# B&R Automation Studio project Kesim (part 2)

#### FbFileCreate.st - File oluşturur.
```iecst
(********************************************************************
 * COPYRIGHT --  B&R Industrial Automation GmbH
 ********************************************************************
 * Library: aLibFile
 * Function Block: FbFileCreate
 * Author: kay3a
 * Created: August 27, 2024/4:58 PM
 ********************************************************************
 * Description: Bu FB secili DeviceName altinda bulunan foler içerisine file olusturur.
 ********************************************************************)
FUNCTION_BLOCK FbFileCreate

	//|ŻŻŻŻŻŻŻŻŻŻŻŻŻŻŻŻŻŻŻŻŻŻŻŻŻŻŻŻŻŻŻŻŻŻŻŻŻŻŻŻŻŻŻŻŻŻŻŻŻŻŻŻŻŻŻŻŻŻŻŻŻŻŻŻŻŻŻŻŻŻŻŻŻ
	//|               FB ENABLE KONTROLU
	//|_________________________________________________________________________

	(* Enable gelirse FB aktiftir. Gelmiyorsa aktif degildir.  *)
	Active := Enable;

	(* Aktif degilse Step basa gelsin *)
	IF NOT Active THEN
		Internal.Step := stepFileCreate_0_Idle;
	END_IF;
	//|_________________________________________________________________________

	//|ŻŻŻŻŻŻŻŻŻŻŻŻŻŻŻŻŻŻŻŻŻŻŻŻŻŻŻŻŻŻŻŻŻŻŻŻŻŻŻŻŻŻŻŻŻŻŻŻŻŻŻŻŻŻŻŻŻŻŻŻŻŻŻŻŻŻŻŻŻŻŻŻŻ
	//|               CHECK FB ERROR
	//|_________________________________________________________________________

	(* Error check *)
	IF (Internal.FB._FileClose.enable AND Internal.FB._FileClose.status <> ERR_FUB_BUSY AND Internal.FB._FileClose.status <> ERR_OK) THEN
		StatusID := Internal.FB._FileClose.status;
		Internal.Step := stepFileCreate_11_Error;

	ELSIF (Internal.FB._FileCreate.enable AND Internal.FB._FileCreate.status <> ERR_FUB_BUSY AND Internal.FB._FileCreate.status <> ERR_OK AND Internal.FB._FileCreate.status <> fiERR_EXIST) THEN
		StatusID := Internal.FB._FileCreate.status;
		Internal.Step := stepFileCreate_11_Error;
	END_IF;
	//|_________________________________________________________________________

	//|ŻŻŻŻŻŻŻŻŻŻŻŻŻŻŻŻŻŻŻŻŻŻŻŻŻŻŻŻŻŻŻŻŻŻŻŻŻŻŻŻŻŻŻŻŻŻŻŻŻŻŻŻŻŻŻŻŻŻŻŻŻŻŻŻŻŻŻŻŻŻŻŻŻ
	//|               CHECK CMD FB EXECUTE
	//|_________________________________________________________________________

	(* Captured Execute *)
	IF EDGEPOS(Execute) THEN
		Internal.CapturedExecute := TRUE;
	ELSIF NOT Execute OR Error THEN
		Internal.CapturedExecute := FALSE;
	END_IF;
	//|_________________________________________________________________________

	//|=========================================================================
	//|					FILLING PROCESS STATE MACHINE
	//|
	//|
	//|=========================================================================
	CASE Internal.Step OF

		//=======================================================
		stepFileCreate_0_Idle: // Idle
			//=======================================================
			Error := FALSE;
			CommandDone := FALSE;
			CommandBusy := FALSE;
			IF Active THEN
				Internal.Step := stepFileCreate_1_WaitCmd;
			END_IF;
			//=======================================================

			//=======================================================
		stepFileCreate_1_WaitCmd: // Wait Cmd
			//=======================================================
			IF (Internal.CapturedExecute) THEN
				CommandBusy := TRUE;
				Internal.Step := stepFileCreate_2_Create;
			END_IF;
			//=======================================================

			//=======================================================
		stepFileCreate_2_Create: // File Create
			//=======================================================
			Internal.FB._FileCreate.enable := TRUE;
			Internal.FB._FileCreate.pDevice := ADR(Parameters.DeviceName);  (* name of the linked device *)
			Internal.FB._FileCreate.pFile := ADR(Parameters.FileName);  (* name of the file *)
			Internal.FB._FileCreate();  (* call the function*)

			IF Internal.FB._FileCreate.status = ERR_OK THEN  (* fileCreate successful *)
				Internal.Step := stepFileCreate_3_Close;  (* next Step*)
			ELSIF Internal.FB._FileCreate.status = fiERR_EXIST THEN
				Internal.Step := stepFileCreate_10_Done;  (* next Step*)
			ELSIF Internal.FB._FileCreate.status = ERR_FUB_BUSY THEN  (* fileCreate not finished -> redo *)
				(* Busy *)
			ELSE  (* Goto Loc.file.Status.error Step *)
				Internal.Step := stepFileCreate_11_Error;
			END_IF
			//=======================================================

			//=======================================================
		stepFileCreate_3_Close: // File Close
			//=======================================================
			Internal.FB._FileClose.enable := TRUE;
			Internal.FB._FileClose.ident := Internal.FB._FileCreate.ident; (* ident for fileCreate-functionblock*)
			Internal.FB._FileClose;  (* call the function*)

			IF Internal.FB._FileClose.status = ERR_OK THEN  (* fileClose successful *)
				Internal.Step := stepFileCreate_10_Done;  (* next Step*)

			ELSIF Internal.FB._FileClose.status = ERR_FUB_BUSY THEN  (* fileClose not finished -> redo *)
				(* Busy *)
			ELSE  (* Goto Loc.file.Status.error Step *)
				Internal.Step := stepFileCreate_11_Error;
			END_IF
			//=======================================================

			//=======================================================
		stepFileCreate_10_Done: // Done
			//=======================================================
			CommandDone := TRUE;
			IF NOT Execute THEN
				Internal.Step := stepFileCreate_0_Idle;
			END_IF;
			//=======================================================

			//=======================================================
		stepFileCreate_11_Error: // Error
			//=======================================================
			Error := TRUE;
			Internal.FB._FileCreate(enable := FALSE);
			Internal.FB._FileClose(enable := FALSE);
			IF ErrorReset THEN
				StatusID := ERR_OK;
				Internal.Step := stepFileCreate_0_Idle;
			END_IF;
		//=======================================================

	END_CASE;
	//|=========================================================================

END_FUNCTION_BLOCK
```

#### FbFileWrite.st - File a yazar.
```iecst
(********************************************************************
 * COPYRIGHT --  B&R Industrial Automation GmbH
 ********************************************************************
 * Library: aLibFile
 * Function Block: FbFileWrite
 * Author: kay3a
 * Created: August 27, 2024/4:58 PM
 ********************************************************************
 * Description:
 ********************************************************************)
FUNCTION_BLOCK FbFileWrite

	//|ŻŻŻŻŻŻŻŻŻŻŻŻŻŻŻŻŻŻŻŻŻŻŻŻŻŻŻŻŻŻŻŻŻŻŻŻŻŻŻŻŻŻŻŻŻŻŻŻŻŻŻŻŻŻŻŻŻŻŻŻŻŻŻŻŻŻŻŻŻŻŻŻŻ
	//|               FB ENABLE KONTROLU
	//|_________________________________________________________________________

	(* Enable gelirse FB aktiftir. Gelmiyorsa aktif degildir.  *)
	Active := Enable;

	(* Aktif degilse Step basa gelsin *)
	IF NOT Active THEN
		Internal.Step := stepFileWrite_0_Idle;
	END_IF;
	//|_________________________________________________________________________

	//|ŻŻŻŻŻŻŻŻŻŻŻŻŻŻŻŻŻŻŻŻŻŻŻŻŻŻŻŻŻŻŻŻŻŻŻŻŻŻŻŻŻŻŻŻŻŻŻŻŻŻŻŻŻŻŻŻŻŻŻŻŻŻŻŻŻŻŻŻŻŻŻŻŻ
	//|               CHECK FB ERROR
	//|_________________________________________________________________________

	(* Error check *)
	IF (Internal.FB._FileClose.enable AND Internal.FB._FileClose.status <> ERR_FUB_BUSY AND Internal.FB._FileClose.status <> ERR_OK) THEN
		StatusID := Internal.FB._FileClose.status;
		Internal.Step := stepFileWrite_11_Error;

	ELSIF (Internal.FB._FileWriteEx.enable AND Internal.FB._FileWriteEx.status <> ERR_FUB_BUSY AND Internal.FB._FileWriteEx.status <> ERR_OK) THEN
		StatusID := Internal.FB._FileWriteEx.status;
		Internal.Step := stepFileWrite_11_Error;

	ELSIF (Internal.FB._FileOpen.enable AND Internal.FB._FileOpen.status <> ERR_FUB_BUSY AND Internal.FB._FileOpen.status <> ERR_OK) THEN
		StatusID := Internal.FB._FileOpen.status;
		Internal.Step := stepFileWrite_11_Error;
	END_IF;
	//|_________________________________________________________________________

	//|ŻŻŻŻŻŻŻŻŻŻŻŻŻŻŻŻŻŻŻŻŻŻŻŻŻŻŻŻŻŻŻŻŻŻŻŻŻŻŻŻŻŻŻŻŻŻŻŻŻŻŻŻŻŻŻŻŻŻŻŻŻŻŻŻŻŻŻŻŻŻŻŻŻ
	//|               CHECK CMD FB EXECUTE
	//|_________________________________________________________________________

	(* Captured Execute *)
	IF EDGEPOS(Execute) THEN
		Internal.CapturedExecute := TRUE;
	ELSIF NOT Execute OR Error THEN
		Internal.CapturedExecute := FALSE;
	END_IF;
	//|_________________________________________________________________________

	//|=========================================================================
	//|					FILLING PROCESS STATE MACHINE
	//|
	//|
	//|=========================================================================
	CASE Internal.Step OF

		//=======================================================
		stepFileWrite_0_Idle: // Idle
			//=======================================================
			Error := FALSE;
			CommandDone := FALSE;
			CommandBusy := FALSE;
			IF Active THEN
				Internal.Step := stepFileWrite_1_WaitCmd;
			END_IF;
			//=======================================================

			//=======================================================
		stepFileWrite_1_WaitCmd: // Wait Cmd
			//=======================================================
			IF (Internal.CapturedExecute) THEN
				CommandBusy := TRUE;
				Internal.Step := stepFileWrite_2_FileOpen;
			END_IF;
			//=======================================================

			//=======================================================
		stepFileWrite_2_FileOpen: // File Open
			//=======================================================
			Internal.FB._FileOpen.enable := TRUE;
			Internal.FB._FileOpen.pDevice := ADR(Parameters.DeviceName);  (* name of the linked device *)

			Internal.FB._FileOpen.pFile :=  ADR(Parameters.FileName);  (* name of the file *)
			Internal.FB._FileOpen.mode := fiWRITE_ONLY; (* write access *)
			Internal.FB._FileOpen();  (* call the function*)

			IF Internal.FB._FileOpen.status = 0 THEN  (* fileOpen successful *)
				Internal.Step := stepFileWrite_3_Write;  (* next Step*)
			ELSIF Internal.FB._FileOpen.status = ERR_FUB_BUSY THEN  (* fileOpen not finished -> redo *)
				(* Busy *)
			ELSE  (* Goto Loc.file.Status.error Step *)
				Internal.Step := stepFileWrite_11_Error;
			END_IF
			//=======================================================

			//=======================================================
		stepFileWrite_3_Write: // File Write
			//=======================================================
			Internal.FB._FileWriteEx.enable := TRUE;
			Internal.FB._FileWriteEx.option := fiTruncate;
			Internal.FB._FileWriteEx.ident := Internal.FB._FileOpen.ident;
			Internal.FB._FileWriteEx.offset := 0; (* start at the beginning of the file *)
			Internal.FB._FileWriteEx.pSrc := ADR(WriteData);
			Internal.FB._FileWriteEx.len := brsstrlen( ADR(WriteData) );
			Internal.FB._FileWriteEx();  (* call the function*)

			IF Internal.FB._FileWriteEx.status = 0 THEN  (* fileWrite successful *)
				Internal.Step := stepFileWrite_4_FileClose;  (* next Step*)
			ELSIF Internal.FB._FileWriteEx.status = ERR_FUB_BUSY THEN  (* fileWrite not finished -> redo *)
				(* Busy *)
			ELSE  (* Goto Loc.file.Status.error Step *)
				Internal.Step := stepFileWrite_11_Error;
			END_IF
			//=======================================================

			//=======================================================
		stepFileWrite_4_FileClose: // File Close
			//=======================================================
			Internal.FB._FileClose.enable := TRUE;
			Internal.FB._FileClose.ident := Internal.FB._FileOpen.ident; (* ident for fileCreate-functionblock*)
			Internal.FB._FileClose();  (* call the function*)

			IF Internal.FB._FileClose.status = 0 THEN  (* fileClose successful *)
				Internal.Step := stepFileWrite_10_Done;  (* next Step*)

			ELSIF Internal.FB._FileClose.status = ERR_FUB_BUSY THEN  (* fileClose not finished -> redo *)
				(* Busy *)
			ELSE  (* Goto Loc.file.Status.error Step *)
				Internal.Step := stepFileWrite_11_Error;
			END_IF
			//=======================================================

			//=======================================================
		stepFileWrite_10_Done: // Done
			//=======================================================
			CommandDone := TRUE;
			IF NOT Execute THEN
				Internal.Step := stepFileWrite_0_Idle;
			END_IF;
			//=======================================================

			//=======================================================
		stepFileWrite_11_Error: // Error
			//=======================================================
			Error := TRUE;
			Internal.FB._FileOpen(enable := FALSE);
			Internal.FB._FileClose(enable := FALSE);
			Internal.FB._FileWriteEx(enable := FALSE);
			IF ErrorReset THEN
				StatusID := ERR_OK;
				Internal.Step := stepFileWrite_0_Idle;
			END_IF;
		//=======================================================

	END_CASE;
	//|=========================================================================

END_FUNCTION_BLOCK
```

#### FbFileRead.st - File i okur.
```iecst
(********************************************************************
 * COPYRIGHT --  B&R Industrial Automation GmbH
 ********************************************************************
 * Library: aLibFile
 * Function Block: FbFileRead
 * Author: kay3a
 * Created: August 27, 2024/4:58 PM
 ********************************************************************
 * Description: Bu FB file içerisini okur.
 ********************************************************************)
FUNCTION_BLOCK FbFileRead

	//|ŻŻŻŻŻŻŻŻŻŻŻŻŻŻŻŻŻŻŻŻŻŻŻŻŻŻŻŻŻŻŻŻŻŻŻŻŻŻŻŻŻŻŻŻŻŻŻŻŻŻŻŻŻŻŻŻŻŻŻŻŻŻŻŻŻŻŻŻŻŻŻŻŻ
	//|               FB ENABLE KONTROLU
	//|_________________________________________________________________________

	(* Enable gelirse FB aktiftir. Gelmiyorsa aktif degildir.  *)
	Active := Enable;

	(* Aktif degilse Step basa gelsin *)
	IF NOT Active THEN
		Internal.Step := stepFileRead_0_Idle;
	END_IF;
	//|_________________________________________________________________________

	//|ŻŻŻŻŻŻŻŻŻŻŻŻŻŻŻŻŻŻŻŻŻŻŻŻŻŻŻŻŻŻŻŻŻŻŻŻŻŻŻŻŻŻŻŻŻŻŻŻŻŻŻŻŻŻŻŻŻŻŻŻŻŻŻŻŻŻŻŻŻŻŻŻŻ
	//|               CHECK FB ERROR
	//|_________________________________________________________________________

	(* Error check *)
	IF (Internal.FB._FileClose.enable AND Internal.FB._FileClose.status <> ERR_FUB_BUSY AND Internal.FB._FileClose.status <> ERR_OK) THEN
		StatusID := Internal.FB._FileClose.status;
		Internal.Step := stepFileRead_11_Error;

	ELSIF (Internal.FB._FileReadEx.enable AND Internal.FB._FileReadEx.status <> ERR_FUB_BUSY AND Internal.FB._FileReadEx.status <> ERR_OK) THEN
		StatusID := Internal.FB._FileReadEx.status;
		Internal.Step := stepFileRead_11_Error;

	ELSIF (Internal.FB._FileOpen.enable AND Internal.FB._FileOpen.status <> ERR_FUB_BUSY AND Internal.FB._FileOpen.status <> ERR_OK) THEN
		StatusID := Internal.FB._FileOpen.status;
		Internal.Step := stepFileRead_11_Error;
	END_IF;
	//|_________________________________________________________________________

	//|ŻŻŻŻŻŻŻŻŻŻŻŻŻŻŻŻŻŻŻŻŻŻŻŻŻŻŻŻŻŻŻŻŻŻŻŻŻŻŻŻŻŻŻŻŻŻŻŻŻŻŻŻŻŻŻŻŻŻŻŻŻŻŻŻŻŻŻŻŻŻŻŻŻ
	//|               CHECK CMD FB EXECUTE
	//|_________________________________________________________________________

	(* Captured Execute *)
	IF EDGEPOS(Execute) THEN
		Internal.CapturedExecute := TRUE;
	ELSIF NOT Execute OR Error THEN
		Internal.CapturedExecute := FALSE;
	END_IF;

	//|_________________________________________________________________________

	//|=========================================================================
	//|					FILLING PROCESS STATE MACHINE
	//|
	//|
	//|=========================================================================
	CASE Internal.Step OF

		//=======================================================
		stepFileRead_0_Idle: // Idle
			//=======================================================
			Error := FALSE;
			CommandDone := FALSE;
			CommandBusy := FALSE;
			IF Active THEN
				Internal.Step := stepFileRead_1_WaitCmd;
			ELSE
				brsmemset(ADR(ReadData), 0, SIZEOF(ReadData));
			END_IF;
			//=======================================================

			//=======================================================
		stepFileRead_1_WaitCmd: // Wait Cmd
			//=======================================================
			IF (Internal.CapturedExecute) THEN
				CommandBusy := TRUE;
				Internal.Step := stepFileRead_2_FileOpen;
			END_IF;
			//=======================================================

			//=======================================================
		stepFileRead_2_FileOpen: // File Open
			//=======================================================
			Internal.FB._FileOpen.enable := TRUE;
			Internal.FB._FileOpen.pDevice := ADR(Parameters.DeviceName);  (* name of the linked device *)

			Internal.FB._FileOpen.pFile :=  ADR(Parameters.FileName);  (* name of the file *)
			Internal.FB._FileOpen.mode := fiREAD_ONLY; (* write access *)
			Internal.FB._FileOpen();  (* call the function*)

			IF Internal.FB._FileOpen.status = 0 THEN  (* fileOpen successful *)
				brsmemset(ADR(ReadData), 0, SIZEOF(ReadData));
				Internal.Step := stepFileRead_3_Read;  (* next Step*)
			ELSIF Internal.FB._FileOpen.status = ERR_FUB_BUSY THEN  (* fileOpen not finished -> redo *)
				(* Busy *)
			ELSE  (* Goto Loc.file.Status.error Step *)
				Internal.Step := stepFileRead_11_Error;
			END_IF
			//=======================================================

			//=======================================================
		stepFileRead_3_Read: // File read
			//=======================================================
			Internal.FB._FileReadEx.enable := TRUE;
			Internal.FB._FileReadEx.ident := Internal.FB._FileOpen.ident;  (* ident of the previous "fileOpen" *)
			Internal.FB._FileReadEx.offset := 0;  (* start at the beginning of the file *)
			Internal.FB._FileReadEx.pDest := ADR(ReadData);  (* adress of the destination of reaaded datas *)
			Internal.FB._FileReadEx.len := SIZEOF(ReadData);  (* lenght of data, which should be readed *)
			Internal.FB._FileReadEx;  (* call the function*)

			IF Internal.FB._FileReadEx.status = 0 THEN  (* fileReadEx successful *)
				(* Internal.FB._FileReadEx.bytesread includes the lenght of the readed data *)
				Internal.Step := stepFileRead_4_FileClose;  (* next Step*)
			ELSIF Internal.FB._FileReadEx.status = ERR_FUB_BUSY THEN  (* fileReadEx not finished -> redo *)
				(* Busy *)
			ELSE  (* Goto Loc.file.Status.error Step *)
				Internal.Step := stepFileRead_11_Error;
			END_IF
			//=======================================================

			//=======================================================
		stepFileRead_4_FileClose: // File Close
			//=======================================================
			Internal.FB._FileClose.enable := TRUE;
			Internal.FB._FileClose.ident := Internal.FB._FileOpen.ident; (* ident for fileCreate-functionblock*)
			Internal.FB._FileClose();  (* call the function*)

			IF Internal.FB._FileClose.status = 0 THEN  (* fileClose successful *)
				Internal.Step := stepFileRead_10_Done;  (* next Step*)

			ELSIF Internal.FB._FileClose.status = ERR_FUB_BUSY THEN  (* fileClose not finished -> redo *)
				(* Busy *)
			ELSE  (* Goto Loc.file.Status.error Step *)
				Internal.Step := stepFileRead_11_Error;
			END_IF
			//=======================================================

			//=======================================================
		stepFileRead_10_Done: // Done
			//=======================================================
			CommandDone := TRUE;
			IF NOT Execute THEN
				Internal.Step := stepFileRead_0_Idle;
			END_IF;
			//=======================================================

			//=======================================================
		stepFileRead_11_Error: // Error
			//=======================================================
			Error := TRUE;
			Internal.FB._FileOpen(enable := FALSE);
			Internal.FB._FileClose(enable := FALSE);
			Internal.FB._FileReadEx(enable := FALSE);
			IF ErrorReset THEN
				StatusID := ERR_OK;
				Internal.Step := stepFileRead_0_Idle;
			END_IF;
		//=======================================================

	END_CASE;
	//|=========================================================================

END_FUNCTION_BLOCK
```

#### FbFileDelete.st - File i siler.
```iecst
(********************************************************************
 * COPYRIGHT --  B&R Industrial Automation GmbH
 ********************************************************************
 * Library: aLibFile
 * Function Block: FbFileDelete
 * Author: kay3a
 * Created: August 27, 2024/4:58 PM
 ********************************************************************
 * Description:
 ********************************************************************)
FUNCTION_BLOCK FbFileDelete

	//|ŻŻŻŻŻŻŻŻŻŻŻŻŻŻŻŻŻŻŻŻŻŻŻŻŻŻŻŻŻŻŻŻŻŻŻŻŻŻŻŻŻŻŻŻŻŻŻŻŻŻŻŻŻŻŻŻŻŻŻŻŻŻŻŻŻŻŻŻŻŻŻŻŻ
	//|               FB ENABLE KONTROLU
	//|_________________________________________________________________________

	(* Enable gelirse FB aktiftir. Gelmiyorsa aktif degildir.  *)
	Active := Enable;

	(* Aktif degilse Step basa gelsin *)
	IF NOT Active THEN
		Internal.Step := stepFileDelete_0_Idle;
	END_IF;
	//|_________________________________________________________________________

	//|ŻŻŻŻŻŻŻŻŻŻŻŻŻŻŻŻŻŻŻŻŻŻŻŻŻŻŻŻŻŻŻŻŻŻŻŻŻŻŻŻŻŻŻŻŻŻŻŻŻŻŻŻŻŻŻŻŻŻŻŻŻŻŻŻŻŻŻŻŻŻŻŻŻ
	//|               CHECK FB ERROR
	//|_________________________________________________________________________

	(* Error check *)
	IF (Internal.FB._FileDelete.enable AND Internal.FB._FileDelete.status <> ERR_FUB_BUSY AND Internal.FB._FileDelete.status <> ERR_OK) THEN
		StatusID := Internal.FB._FileDelete.status;
		Internal.Step := stepFileDelete_11_Error;
	END_IF;
	//|_________________________________________________________________________

	//|ŻŻŻŻŻŻŻŻŻŻŻŻŻŻŻŻŻŻŻŻŻŻŻŻŻŻŻŻŻŻŻŻŻŻŻŻŻŻŻŻŻŻŻŻŻŻŻŻŻŻŻŻŻŻŻŻŻŻŻŻŻŻŻŻŻŻŻŻŻŻŻŻŻ
	//|               CHECK CMD FB EXECUTE
	//|_________________________________________________________________________

	(* Captured Execute *)
	IF EDGEPOS(Execute) THEN
		Internal.CapturedExecute := TRUE;
	ELSIF NOT Execute OR Error THEN
		Internal.CapturedExecute := FALSE;
	END_IF;
	//|_________________________________________________________________________

	//|=========================================================================
	//|					FILLING PROCESS STATE MACHINE
	//|
	//|
	//|=========================================================================
	CASE Internal.Step OF

		//=======================================================
		stepFileDelete_0_Idle: // Idle
			//=======================================================
			Error := FALSE;
			CommandDone := FALSE;
			CommandBusy := FALSE;
			IF Active THEN
				Internal.Step := stepFileDelete_1_WaitCmd;
			END_IF;
			//=======================================================

			//=======================================================
		stepFileDelete_1_WaitCmd: // Wait Cmd
			//=======================================================
			IF (Internal.CapturedExecute) THEN
				CommandBusy := TRUE;
				Internal.Step := stepFileDelete_2_Delete;
			END_IF;
			//=======================================================

			//=======================================================
		stepFileDelete_2_Delete: // Delete
			//=======================================================
			Internal.FB._FileDelete.enable := TRUE;
			Internal.FB._FileDelete.pDevice := ADR(Parameters.DeviceName);  (* name of a linked device *)

			Internal.FB._FileDelete.pName := ADR(Parameters.FileName);  (* name of the source file *)
			Internal.FB._FileDelete;  (* call the function*)

			IF Internal.FB._FileDelete.status = 0 THEN  (* filedelete successful *)
				Internal.Step := stepFileDelete_10_Done;  (* next Step*)

			ELSIF Internal.FB._FileDelete.status = ERR_FUB_BUSY THEN  (* fileDelete not finished -> redo *)
				(* Busy *)
			ELSE  (* Goto Loc.file.Status.error Step *)
				Internal.Step := stepFileDelete_11_Error;
			END_IF
			//=======================================================

			//=======================================================
		stepFileDelete_10_Done: // Done
			//=======================================================
			CommandDone := TRUE;
			IF NOT Execute THEN
				Internal.Step := stepFileDelete_0_Idle;
			END_IF;
			//=======================================================

			//=======================================================
		stepFileDelete_11_Error: // Error
			//=======================================================
			Error := TRUE;
			Internal.FB._FileDelete(enable := FALSE);
			IF ErrorReset THEN
				StatusID := ERR_OK;
				Internal.Step := stepFileDelete_0_Idle;
			END_IF;
		//=======================================================

	END_CASE;
	//|=========================================================================

END_FUNCTION_BLOCK
```

### Library Logical/Libraries/CMS_CT (IEC)

#### Types.typ - Exported data types
```iecst
TYPE
	MachineTypes_Enm :
		(
		OCKM := 0,
		FCL := 1,
		FCM := 2,
		YCKM := 3
		);
END_TYPE
```

#### fbTableUpDown.typ
```iecst
TYPE
	fbTableUpDownInCmd_type : 	STRUCT
		Up : BOOL;
		Down : BOOL;
		Error : BOOL;
		Pause : BOOL;
		Reset : BOOL;
		Stop : BOOL;
	END_STRUCT;
	fbTableUpDownOut_type : 	STRUCT
		Hyd : fbTableUpDownOutHyd_type;
		ReadyToCut : BOOL;
		Stoped : BOOL;
		CommandDone : USINT;
		CommandBusy : USINT;
		ErrorID : fbTableUpDownErrorID_enm;
		Error : BOOL;
	END_STRUCT;
	fbTableUpDownInSensors_type : 	STRUCT
		TableDownSlow : BOOL;
		TableUpSlow : BOOL;
		TableIsDown : BOOL;
		TableSquaresAreBack : BOOL;
		TableIsUp : BOOL;
		TableMotFault : BOOL;
	END_STRUCT;
	fbTableUpDownOutHyd_type : 	STRUCT
		BypassValve : BOOL;
		DownValve : BOOL;
		DownSlow : BOOL;
		UpValve : BOOL;
		UpSlowValve : BOOL;
		HydStart : BOOL;
	END_STRUCT;
	fbTableUpDownIn_type : 	STRUCT
		Sensors : fbTableUpDownInSensors_type;
		HomingDone : BOOL;
		ParkPos : BOOL;
		Cmd : fbTableUpDownInCmd_type;
	END_STRUCT;
	fbTableUpDownErrorID_enm :
		(
		ERR_NONE := 0,
		SQUARES_ARE_NOT_DOWN := 10,
		SQUARES_ARE_NOT_UP := 20,
		MACHINE_IS_NOT_PARK_POS := 30,
		TABLE_IS_NOT_DOWN := 40,
		HOMING_IS_REQUIRED := 50,
		TABLE_MOTOR_FAULT := 60
		);
END_TYPE
```

#### CMS_CT.fun - Exported functions and function blocks
```iecst
{REDUND_ERROR} {REDUND_UNREPLICABLE} FUNCTION_BLOCK fbTONOF (*TON And TOF Timer*) (*$GROUP=User,$CAT=User,$GROUPICON=User.png,$CATICON=User.png*)
	VAR_INPUT
		Input : {REDUND_UNREPLICABLE} BOOL;
		TON_Time : {REDUND_UNREPLICABLE} TIME;
		TOF_Time : {REDUND_UNREPLICABLE} TIME;
	END_VAR
	VAR_OUTPUT
		Q : {REDUND_UNREPLICABLE} BOOL;
	END_VAR
	VAR
		mode : {REDUND_UNREPLICABLE} BOOL;
		old : {REDUND_UNREPLICABLE} BOOL;
		TON_Timer : {REDUND_UNREPLICABLE} TON;
	END_VAR
END_FUNCTION_BLOCK

{REDUND_ERROR} FUNCTION_BLOCK fbToggle (*TODO: Toggle*) (*$GROUP=User,$CAT=User,$GROUPICON=User.png,$CATICON=User.png*)
	VAR_INPUT
		Enable : BOOL;
		CLK : {REDUND_UNREPLICABLE} BOOL;
		Rst : {REDUND_UNREPLICABLE} BOOL;
	END_VAR
	VAR_OUTPUT
		Q : {REDUND_UNREPLICABLE} BOOL;
	END_VAR
	VAR
		_edge : {REDUND_UNREPLICABLE} BOOL;
	END_VAR
END_FUNCTION_BLOCK

FUNCTION_BLOCK fbStateHistory (*State History LOgger*) (*$GROUP=User,$CAT=User,$GROUPICON=User.png,$CATICON=User.png*)
	VAR_INPUT
		inEnable : {REDUND_UNREPLICABLE} BOOL;
		inReset : {REDUND_UNREPLICABLE} BOOL;
		inAlarm : BOOL;
		inActState : {REDUND_UNREPLICABLE} INT;
		N : {REDUND_UNREPLICABLE} INT;
	END_VAR
	VAR_OUTPUT
		outStateHistory : {REDUND_UNREPLICABLE} ARRAY[0..10] OF INT;
		outErrorHistory : ARRAY[0..2,0..10] OF INT;
	END_VAR
	VAR
		OldActState : {REDUND_UNREPLICABLE} INT;
		j : {REDUND_UNREPLICABLE} INT;
		i : {REDUND_UNREPLICABLE} INT;
	END_VAR
END_FUNCTION_BLOCK

{REDUND_ERROR} FUNCTION_BLOCK fbTableUpDown (*Table Up Down Movement for OCKM And Breaker*) (*$GROUP=User,$CAT=User,$GROUPICON=User.png,$CATICON=User.png*)
	VAR_INPUT
		Enable : BOOL;
		In : {REDUND_UNREPLICABLE} fbTableUpDownIn_type;
	END_VAR
	VAR_OUTPUT
		Out : {REDUND_UNREPLICABLE} fbTableUpDownOut_type;
	END_VAR
	VAR
		OldStep : UINT;
		FirstInStep : BOOL;
		TOF_Hyd : TOF;
		Step : UINT;
	END_VAR
END_FUNCTION_BLOCK
```

#### fbToggle.st
```iecst
(* TODO: Toggle *)
FUNCTION_BLOCK fbToggle

IF Enable THEN

	IF Rst THEN
		Rst := 0;
		Q 	:= 0;
	ELSIF CLK AND NOT _edge THEN
		Q := NOT Q;
	END_IF;
ELSE
	Q 	:= 0;
END_IF
 _edge := CLK;
END_FUNCTION_BLOCK
```

#### fbTONOF.st
```iecst
(* TON And TOF Timer *)
FUNCTION_BLOCK fbTONOF

	IF Input  XOR old THEN
		TON_Timer(IN:=FALSE , PT:= SEL(Input, TOF_Time, TON_Time ));
		mode	 := Input;
		old		 := Input;
	END_IF;

	TON_Timer( IN := TRUE);

	IF TON_Timer.Q THEN
		Q := mode;
	END_IF;

END_FUNCTION_BLOCK
```

#### fbStateHistory.st
```iecst
(* State History LOgger *)
FUNCTION_BLOCK fbStateHistory

	IF inReset THEN

		FOR i:=0 TO N DO
			outStateHistory[i]:= 0;
			inReset	:= FALSE;
		END_FOR

	ELSIF inActState <> OldActState THEN

		FOR i:= N TO 1 BY -1 DO
			outStateHistory[i] := outStateHistory[i-1];
		END_FOR
		outStateHistory[0] := inActState;

		IF inAlarm THEN // bc25.07.14
			//			outErrorHistory := outStateHistory;

			FOR i:= N TO 1 BY -1 DO
				outErrorHistory[2,i] := outErrorHistory[1,i];
				outErrorHistory[1,i] := outErrorHistory[0,i];
				outErrorHistory[0,i] := outStateHistory[i];
			END_FOR

		END_IF

	END_IF
	OldActState := inActState;

END_FUNCTION_BLOCK
```

#### fbTableUpDown.st
```iecst
(* Table Up Down Movement for OCKM And Breaker *)
FUNCTION_BLOCK fbTableUpDown

	IF Enable = FALSE THEN
		brsmemset( ADR(Out.Hyd),0,SIZEOF(Out.Hyd) );
		Out.ReadyToCut  := FALSE;
		Step			:= 0;
		RETURN;
	ELSE

		IF In.Sensors.TableMotFault THEN
			Step 		:= 999;
			Out.ErrorID := TABLE_MOTOR_FAULT;
		END_IF;

		IF In.Cmd.Stop AND NOT Out.Error THEN
			Step		:= 50;
		END_IF;

		//|ŻŻŻŻŻŻŻŻŻŻŻŻŻŻŻŻŻŻŻŻŻŻŻŻŻŻŻŻŻŻŻŻŻŻŻŻŻŻŻŻŻŻŻŻŻŻŻŻŻŻŻŻŻŻŻŻŻŻŻŻŻŻŻŻŻŻŻŻŻŻŻŻŻ
		//|               Table Is Ready To Cut
		//|_________________________________________________________________________
		Out.ReadyToCut :=
		In.Sensors.TableSquaresAreBack AND In.Sensors.TableIsDown AND
		In.ParkPos AND NOT In.Sensors.TableIsUp AND
		NOT In.Sensors.TableUpSlow AND In.ParkPos;

		CASE Step OF
			0: // INIT
				Out.Error 	:= FALSE;
				Out.ErrorID := ERR_NONE;
				Out.Stoped 	:= FALSE;
				brsmemset( ADR(Out.Hyd),0,SIZEOF(Out.Hyd) );
				Step 		:= 10;
			10:
				IF In.Cmd.Up OR In.Cmd.Down  THEN
					IF In.Sensors.TableSquaresAreBack THEN
						Step 		:= 999;
						Out.ErrorID := SQUARES_ARE_NOT_UP;
						RETURN;
					ELSIF In.HomingDone = FALSE THEN
						Step 		:= 999;
						Out.ErrorID := HOMING_IS_REQUIRED;
						RETURN;
					ELSIF In.ParkPos = FALSE THEN
						Step 		:= 999;
						Out.ErrorID := MACHINE_IS_NOT_PARK_POS;
						RETURN;
					ELSE
						// Command Active
						IF In.Cmd.Up THEN
							Step		:= 20;
						ELSIF In.Cmd.Down THEN
							Step		:= 30;
						END_IF;
					END_IF;

				END_IF;

			20: // Command Up
				IF 	In.Cmd.Up = FALSE THEN
					Step 		:= 0;
				ELSE
					IF 	In.Sensors.TableIsUp THEN
						Out.Hyd.UpSlowValve := FALSE;
						Out.Hyd.UpValve     := FALSE;
						Step 				:= 40; // Command Done
					ELSIF In.Sensors.TableUpSlow THEN
						Out.Hyd.UpValve  	:= TRUE;
						Out.Hyd.UpSlowValve := TRUE;
					ELSE
						Out.Hyd.UpValve  	:= TRUE;
						Out.Hyd.UpSlowValve := FALSE;
					END_IF;
				END_IF;

			30: // Command Down
				IF 	In.Cmd.Down = FALSE THEN
					Step 		:= 0;
				ELSE
					IF 	In.Sensors.TableIsDown THEN
						Out.Hyd.DownSlow	:= FALSE;
						Out.Hyd.DownValve   := FALSE;
						Step 				:= 40; // Command Done
					ELSIF In.Sensors.TableDownSlow THEN
						Out.Hyd.DownSlow	:= TRUE;
						Out.Hyd.DownValve  := TRUE;
					ELSE
						Out.Hyd.DownSlow	:= TRUE;
						Out.Hyd.DownValve  := FALSE;
					END_IF;
				END_IF;

			40: // Command Done
				Out.CommandDone := TRUE;
				brsmemset( ADR(Out.Hyd),0,SIZEOF(Out.Hyd) );

				IF NOT In.Cmd.Down AND
					NOT In.Cmd.Up AND
					NOT In.Cmd.Pause AND
					NOT In.Cmd.Stop THEN
					Step := 0;
				END_IF;

			50: // Stop Command
				Out.Stoped 		:= TRUE;
				brsmemset( ADR(Out.Hyd),0,SIZEOF(Out.Hyd) );
				Step 			:= 40; // Command Done

			999:
				Out.Error := TRUE;
				brsmemset( ADR(Out.Hyd),0,SIZEOF(Out.Hyd) );
				Out.ReadyToCut  := FALSE;
				IF In.Cmd.Reset THEN
					Step := 0;
				END_IF;

		END_CASE;

		// Hydraulic Motor Output
		TOF_Hyd.IN 		:= Out.Hyd.UpValve OR Out.Hyd.DownValve OR Out.Hyd.UpSlowValve OR Out.Hyd.UpSlowValve ;
		TOF_Hyd.PT 		:= T#3s;
		Out.Hyd.HydStart := TOF_Hyd.Q;

		TOF_Hyd();

	END_IF;

	FirstInStep := OldStep <> Step;
	OldStep 	:= Step;

END_FUNCTION_BLOCK
```

#### fbCuttingTransfer.st
```iecst
(* Transfer Glass To Cutting OR To Breaker *)
FUNCTION_BLOCK fbCuttingTransfer

		//==============================
	//		FB Enable Check
	//==============================
	IF inEnable THEN
		outActive := TRUE;
	ELSE
		outActive 		:= FALSE;
		outError		:= FALSE;
		outErrorID		:= NO_ERROR;
		outState		:= CT_INIT;
		brsmemset(ADR(outDO), 0, SIZEOF(outDO));
		brsmemset(ADR(Loc), 0, SIZEOF(Loc));
		brsmemset(ADR(inSensors), 0, SIZEOF(inSensors));
		RETURN;
	END_IF;
	//==============================

	//State Timer
	Loc.StepTimer();

	// Error ID ler yazilacak
	outGlassTransferActive := (Loc.GlassTransferActive OR Loc.GlassGettingActive);

	CASE outState OF
		CT_INIT:
			outError				:= FALSE;
			outErrorID				:= NO_ERROR;
			brsmemset(ADR(outDO), 0, SIZEOF(outDO));
			brsmemset(ADR(Loc), 0, SIZEOF(Loc));
			inGlassTransfer 		:= FALSE;
			outGlassTransferDone 	:= FALSE;
			outGlassTransferActive	:= FALSE;
			outCommandDone			:= FALSE;
			Loc.StepTimer.IN 		:= FALSE;
			outState				:= CT_WAIT_CMD;

		CT_WAIT_CMD:

			IF      inGlassTransfer AND inCTReadyToTransfer
				AND inLoaderReadyToTransfer AND NOT inSensors.BeltStop_SW
				AND NOT Loc.GlassGettingActive AND NOT Loc.GlassTransferActive THEN
				outState				:= CT_BELT_UP;
				Loc.GlassGettingActive 	:= TRUE;
			END_IF

			IF      inGlassTransfer AND inCTReadyToTransfer
				AND  inSensors.BeltStop_SW AND inSensors.BT_DownSW
				AND NOT Loc.GlassGettingActive AND NOT Loc.GlassTransferActive  THEN
				outState			 	:= CT_BELT_UP;
				Loc.GlassTransferActive := TRUE;
				outDO.BT_FanStart  		:= TRUE;
			END_IF;

		CT_BELT_UP: 	(***********WAIT BELT UP FOR CT TRANSFER MOTOR START******************)
			IF Loc.FirstInStep THEN
				outDO.CT_TransportBeltUp 	:= TRUE;
				outDO.CT_YCARRIERDOWNVALVE 	:= FALSE;
				Loc.StepTimer.PT 			:= T#5000ms;
				Loc.StepTimer.IN			:= TRUE;
			ELSE
				IF 	inSensors.YCarrBack_SW AND inSensors.BeltUp_SW THEN
					Loc.StepTimer.IN := FALSE;
					outDO.CT_GLASSTRANSPORTMOTORSTART := TRUE;
					outState 						  := CT_GET_OR_TRANSFER_GLASS;
				END_IF;
			END_IF;

			IF inSimulation THEN
				IF Loc.StepTimer.Q THEN
					Loc.StepTimer(IN:= FALSE);
				ELSIF Loc.StepTimer.ET >= T#2000ms THEN
					// Belt Is Up
					inSensors.BeltUp_SW		:= TRUE;
					inSensors.BeltDown_SW 	:= FALSE;
				ELSIF Loc.StepTimer.ET >= T#200ms THEN
					// Belt Still Down
					inSensors.BeltUp_SW		:= FALSE;
					inSensors.BeltDown_SW 	:= TRUE;
				END_IF;
			END_IF

		CT_GET_OR_TRANSFER_GLASS:

			IF Loc.GlassGettingActive  THEN
				outDO.L_GLASSTRANSPORTSTART := TRUE;
				outState := CT_WAIT_FINISH_TRANS;
			ELSIF Loc.GlassTransferActive THEN
				outDO.L_GLASSTRANSPORTSTART := FALSE;
				outState := CT_WAIT_FINISH_TRANS;
			END_IF;

		CT_WAIT_FINISH_TRANS:
			IF Loc.GlassGettingActive AND inSensors.BeltStop_SW THEN
				outDO.L_GLASSTRANSPORTSTART 		:= FALSE;
				outDO.CT_GLASSTRANSPORTMOTORSTART 	:= FALSE;

				Loc.StepTimer.IN 			:= TRUE;
				Loc.StepTimer.PT 			:= T#5s;
				// Wait Belt Stop Down Ramp
				IF Loc.StepTimer.Q THEN
					Loc.StepTimer.IN 		:= FALSE;
					outState 				:= CT_BELT_DOWN;
				END_IF
			ELSIF Loc.GlassGettingActive AND NOT inSensors.BeltStop_SW AND NOT inSensors.BeltGlassExit_SW AND NOT inLoaderReadyToTransfer THEN
				outDO.L_GLASSTRANSPORTSTART 		:= FALSE;
				outDO.CT_GLASSTRANSPORTMOTORSTART 	:= FALSE;
				outState 							:= CT_BELT_DOWN;
			ELSIF Loc.GlassTransferActive AND NOT inSensors.BeltStop_SW AND NOT inSensors.BeltGlassExit_SW AND inLoaderReadyToTransfer  THEN
				Loc.GlassTransferActive 			:= FALSE;
				Loc.GlassGettingActive  			:= TRUE;
				outState 							:= CT_BELT_UP;
			ELSIF Loc.GlassTransferActive AND NOT inSensors.BeltStop_SW AND NOT inSensors.BeltGlassExit_SW AND NOT inLoaderReadyToTransfer  THEN
				Loc.GlassTransferActive 			:= FALSE;
				Loc.GlassGettingActive  			:= TRUE;
				outState 							:= CT_BELT_DOWN;
			END_IF;

			IF Loc.GlassGettingActive AND NOT Loc.LoaderGlassExitDelay.Q THEN
				outDO.L_GLASSTRANSPORTSTART 		:= FALSE;
			END_IF;

		CT_BELT_DOWN:

			IF Loc.FirstInStep THEN
				Loc.StepTimer.IN 			:= TRUE;
				Loc.StepTimer.PT 			:= T#5s;
				outDO.CT_TransportBeltUp 	:= FALSE;
			ELSE
				IF Loc.TON_BeltDown.Q THEN
					outState := CT_WAIT_CMD_DONE;

				ELSIF Loc.StepTimer.Q AND NOT inSimulation THEN
					outState 			:= CT_TRANS_ERROR;
					outErrorID			:= CT_BELT_IS_NOT_DOWN;

				END_IF;
			END_IF

			IF inSimulation THEN
				IF Loc.StepTimer.Q THEN
					Loc.StepTimer(IN:= FALSE);
				ELSIF Loc.StepTimer.ET >= T#2000ms THEN
					// Belt Is Up
					inSensors.BeltUp_SW		:= FALSE;
					inSensors.BeltDown_SW 	:= TRUE;
				ELSIF Loc.StepTimer.ET >= T#200ms THEN
					// Belt Still Down
					inSensors.BeltUp_SW		:= TRUE;
					inSensors.BeltDown_SW 	:= FALSE;
				END_IF;
			END_IF

		CT_WAIT_CMD_DONE:
			IF Loc.FirstInStep THEN
				outCommandDone := TRUE;
				Loc.StepTimer.IN := FALSE;
			ELSE
				IF NOT inGlassTransfer THEN
					// Waiting fb Input cmd's are OFF
					outState := CT_INIT;
				END_IF;
			END_IF;

		CT_TRANS_ERROR:
			IF Loc.FirstInStep THEN
				brsmemset(ADR(outDO), 0, SIZEOF(outDO));
				outError 	:= TRUE;
				Loc.StepTimer(IN:= FALSE);
			ELSE
				IF inReset THEN
					outErrorID := CT_BELT_IS_NOT_DOWN;
					outState := CT_INIT;
				END_IF;
			END_IF;

	END_CASE;

	// Errors
	IF inSensors.CT_BeltMotFault THEN
		outErrorID := CT_TRANS_BELT_MOT_FAULT;
		outState   := CT_TRANS_ERROR;
	END_IF;

	// Timers
	// Glass Exit TOF Delay
	Loc.LoaderGlassExitDelay.IN := inSensors.BeltGlassExit_SW;
	Loc.LoaderGlassExitDelay.PT := T#1.5s;
	Loc.LoaderGlassExitDelay();

	// Belt Down TON Delay
	Loc.TON_BeltDown.IN := NOT outDO.CT_TransportBeltUp AND inSensors.BeltDown_SW;
	Loc.TON_BeltDown.PT := T#1s;
	Loc.TON_BeltDown();

	// First In Step Control
	IF (outState <> Loc.OldState) THEN
		Loc.FirstInStep := TRUE;
	ELSE
		Loc.FirstInStep := FALSE;
	END_IF;
	Loc.OldState 	:= outState;

END_FUNCTION_BLOCK
```

#### fbCuttingTransfer.typ - not listed in the package file held
```iecst
TYPE
	fbCuttingTransferLoc_type : 	STRUCT
		GlassGettingActive : BOOL;
		GlassTransferActive : BOOL;
		FirstInStep : BOOL;
		OldState : fbCuttingTransferState_type;
		TON_BeltDown : TON;
		LoaderGlassExitDelay : TOF;
		StepTimer : TON;
	END_STRUCT;
	fbCuttingTransferSens_type : 	STRUCT
		LoaderGlassExit_SW : BOOL;
		BeltGlassExit_SW : BOOL;
		BeltStop_SW : BOOL;
		BeltUp_SW : BOOL;
		BeltDown_SW : BOOL;
		BT_DownSW : BOOL;
		YCarrBack_SW : BOOL;
		CT_BeltMotFault : BOOL;
	END_STRUCT;
	fbCuttingTransferState_type :
		(
		CT_INIT := -1,
		CT_WAIT_CMD := 0,
		CT_BELT_UP := 1,
		CT_GET_OR_TRANSFER_GLASS := 2,
		CT_WAIT_FINISH_TRANS := 3,
		CT_BELT_DOWN := 4,
		CT_WAIT_BELT_DOWN := 5,
		CT_WAIT_CMD_DONE := 6,
		CT_TRANS_ERROR := 999
		);
	fbCuttingTransferDO_type : 	STRUCT
		GlassTransToCuttingTable : BOOL;
		CT_TransportBeltUp : BOOL;
		CT_YCARRIERDOWNVALVE : BOOL;
		CT_GLASSTRANSPORTMOTORSTART : BOOL;
		L_GLASSTRANSPORTSTART : BOOL;
		BT_FanStart : BOOL; (*Breaker Table Fan Start*)
	END_STRUCT;
	fbCuttingTransfeErrorID_type :
		(
		NO_ERROR := 0,
		CT_TRANS_BELT_MOT_FAULT,
		CT_BELT_IS_NOT_DOWN
		);
END_TYPE
```

#### fcFind_Origin.st
```iecst
(* The equation of a line where 2 points are known and the 3rd point is perpendicular to it. *)
FUNCTION fcFind_Origin

IF Enable THEN

	m2		:= (Y2 - Y1) / (X2 - X1);	// Iki noktasi okunan dogrunun egimi
	F_LIN2 	:= m2 * (X - X1) + Y1;  	// Iki noktasi okunan dogrunun denklemi
	m1     	:= -1/m2;			    	// Bir noktasi okunan dogrunun egimi
	F_LIN1 	:= m1 * (X - X3) + Y3;  	// Bir noktasi okunan ve egimi bilinen dogru denklemi

	k		:= ATAN(m2);					  // Hesaplama
	DEGREE	:= k * 180 / (3.14159265); 		  // Iki noktasi okunan dogrunun X eksenindeki dönüklügünün açi degeri
	RADYAN	:= (DEGREE * (3.14159265)) / 180; // Iki noktasi okunan dogrunun X eksenindeki dönüklügünün açi degeri

	IF m2<>0 THEN

		X0     := ( (Y3-Y1)+(m2*X1)-(m1*X3) ) / (m2-m1);    // Parca Sifiri X degeri
		Y0     := m2 *(X0 - X1)+Y1;							// Parca Sifiri Y degeri
	ELSIF m2=0 THEN // Cam Tam 90 derece konulmus
		X0     := X3 + SearchSensorXOffset;   // Gb_X3:= MC_TouchProbe_X.RecordedPosition + VarHmictrl_Sensor_X; // Ilk Okunan X Noktasinin Offsetli degeri
		Y0     := Y1 + SearchSensorYOffset;   // Gb_Y1:= MC_TouchProbe_Y.RecordedPosition + VarHmictrl_Sensor_Y; // Ikinci Okunan Degerin Y Offsetli degeri
	END_IF;

ELSE // No Enable
	;
END_IF;

	// Y eksen
	//
	//
	////  nokta 3
	//
	//
	//
	//  	nokta 2			nokta 1
	//		//				//
	/////////////////////////////////////// X eksen

END_FUNCTION
```

### Library Logical/Libraries/IOControl (IEC, version 1.0.5) - IO Control Library
Depends on: AsIOMMan, AsIODiag, AsIO

#### IOControl.typ - Exported data types
```iecst
(********************************************************************
 * COPYRIGHT -- Bernecker + Rainer
 ********************************************************************
 * Library: IOControl
 * File: IOControl.typ
 * Author: abdullahoglf
 * Created: February 12, 2014
 ********************************************************************
 * Data types of library IOControl
 ********************************************************************)

TYPE
	IOTypeChannel_enm :
		(
		DI_IO := 0,
		DO_IO := 1,
		AI_IO := 2,
		AO_IO := 3
		);
END_TYPE
```

#### IOControl.fun - Exported functions and function blocks
```iecst
(********************************************************************
 * COPYRIGHT -- Bernecker + Rainer
 ********************************************************************
 * Library: IOControl
 * File: IOControl.fun
 * Author: abdullahoglf
 * Created: February 12, 2014
 ********************************************************************
 * Functions and function blocks of library IOControl
 ********************************************************************)

FUNCTION_BLOCK BuildSignalStr (*Builds the necessary datapoint for a specific channel*)
	VAR_INPUT
		uNumStation : USINT;
		uNumSignal : USINT; (*Channel number*)
		eTypeSignal : IOTypeChannel_enm; (*Channel type*)
		sStrSignal : STRING[255];
		selectedWashingModule : BOOL;
	END_VAR
	VAR
		str : STRING[255];
		sEPL : STRING[32];
	END_VAR
END_FUNCTION_BLOCK
```

#### BuildSignalStr.st - Builds the necessary datapoint for a specific channel
```iecst
(********************************************************************
 * COPYRIGHT -- Bernecker + Rainer
 ********************************************************************
 * Library: IOControl
 * File: BuildSignalStr.st
 * Author: abdullahoglf
 * Created: February 12, 2014
 ********************************************************************
 * Implementation of library IOControl
 ********************************************************************)

(* Builds the necessary datapoint for a specific channel *)
FUNCTION_BLOCK BuildSignalStr

		// build string: step 1 : direction prefix and size prefix
		CASE eTypeSignal OF
			(* --- *)
			DI_IO:
				sStrSignal := '%IX';

				(* --- *)
			DO_IO:
				sStrSignal := '%QX';

				(* --- *)
			AI_IO:
				sStrSignal := '%IW';

				(* --- *)
			AO_IO:
				sStrSignal := '%QW';

		END_CASE;

		(* --- *)
		// build string: step 2 : add powerlink interface name
		brsstrcat(ADR(sStrSignal),ADR(sEPL));

		// num slot
		brsstrcat(ADR(sStrSignal),ADR('.IF6'));

		(* --- *)
		// build string: step 3 : num station and num slot
		// num station
		brsitoa(USINT_TO_DINT(uNumStation), ADR(str));

		brsstrcat(ADR(sStrSignal),ADR('.ST'));
		brsstrcat(ADR(sStrSignal),ADR(str));

		//	itoa(USINT_TO_DINT(uNumSlot), ADR(str));
		//	strcat(ADR(sStrSignal),ADR(str));

		(* --- *)
		// build string: step 4 : channel name
		CASE eTypeSignal OF
			(* --- *)
			DI_IO:
				str := '.DigitalInput';

				(* --- *)
			DO_IO:
				str := '.DigitalOutput';

				(* --- *)
			AI_IO:
				str := '.AnalogInput';

				(* --- *)
			AO_IO:
				str := '.AnalogOutput';
		END_CASE;

		CASE uNumSignal OF

			0: (* this Channel is not configured *);
				str := 'NOT CONFIGURED';

			1:	(* ChannelName01 *)
				brsstrcat(ADR(str),ADR('01'));

			2:	(* ChannelName02 *)
				brsstrcat(ADR(str),ADR('02'));

			3:	(* ChannelName03 *)
				brsstrcat(ADR(str),ADR('03'));

			4: (* ChannelName04 *)
				brsstrcat(ADR(str),ADR('04'));

			5: (* ChannelName05 *)
				brsstrcat(ADR(str),ADR('05'));

			6:	(* ChannelName06 *)
				brsstrcat(ADR(str),ADR('06'));

			7:	(* ChannelName07 *)
				brsstrcat(ADR(str),ADR('07'));

			8:	(* ChannelName08 *)
				brsstrcat(ADR(str),ADR('08'));

			9: (* ChannelName09 *)
				brsstrcat(ADR(str),ADR('09'));

			10:(* ChannelName10 *)
				brsstrcat(ADR(str),ADR('10'));

			11:(* ChannelName11 *)
				brsstrcat(ADR(str),ADR('11'));

			12:(* ChannelName12 *)
				brsstrcat(ADR(str),ADR('12'));

			13:(* ChannelName13 *)
				brsstrcat(ADR(str),ADR('13'));

			14:(* ChannelName14 *)
				brsstrcat(ADR(str),ADR('14'));

			15:(* ChannelName15 *)
				brsstrcat(ADR(str),ADR('15'));

			16:(* ChannelName16 *)
				brsstrcat(ADR(str),ADR('16'));

		END_CASE

		brsstrcat(ADR(sStrSignal),ADR(str));

END_FUNCTION_BLOCK
```

### GlobalAlertConst.var - Global variables
```iecst
(*********************************************************************************
 * Copyright:
 * Author:    baranc
 * Created:   October 21, 2025/8:32 AM
 *********************************************************************************)
(*Genaral Class Error 0..99*)
VAR CONSTANT
	ALERT_E_STOP : UDINT := 0; (*E-stop is pressed*)
	ALERT_PHASE_LOST : UDINT := 1; (*Electrical phase lost detection*)
	ALERT_AIR_SUPLY_ERROR : UINT := 2;
	ALERT_POWER_ON_PROBLEM : UINT := 3;
	ALERT_CONV_ENTRY1 : UINT := 4;
	ALERT_CONV_ENTRY2 : UINT := 5;
	ALERT_CONV_ENTRY3 : UINT := 6;
	ALERT_CONV_ENTRY4 : UINT := 7;
	ALERT_CONV_EXIT1 : UINT := 8;
	ALERT_CONV_EXIT2 : UINT := 9;
	ALERT_CONV_EXIT3 : UINT := 10;
	ALERT_CONV_EXIT4 : UINT := 11;
	ALERT_CONV_EXIT5 : UINT := 12;
	ALERT_CONV_EXIT6 : UINT := 13;
	ALERT_CONV_EXIT7 : UINT := 14;
	ALERT_CONV_EXIT8 : UINT := 15;
	ALERT_HEAD_Y : UINT := 16;
	ALERT_HEAD_C : UINT := 17;
	ALERT_HEAD_Z : UINT := 18;
	ALERT_HYD : UINT := 19;
	ALERT_VACUUM : UINT := 20;
	ALERT_EX1_BRIDGE : UINT := 21;
	ALERT_PARKING_IO_NOT_PARKED : UINT := 22; (*Parking is not possible - Check Inputs and Outputs*)
	ALERT_FILLING_IS_TAKING_TOO_LONG : UINT := 23; (*Filling is taking too long (over 2 minutes)*)
	ALERT_MAT_IN_MIXER_TIME_2ND_ERR : UINT := 24; (*Material in mixer is too long - Make Cleaning or Dossing*)
	ALERT_HOMING_TIMEOUT : UINT := 25;
	ALERT_CZ_ABS_ENC_NOT_ADJUSTED : UINT := 26;
	ALERT_CHECK_GLASS_THICNESS : UINT := 27;
	ALERT_VAC_LIMIT : UINT := 28;
END_VAR
(**)
VAR CONSTANT
	ERR_H_AXIS_IS_NOT_READY_TO_START : UINT := 900; (*Hydr. Axis is not ready to start*)
	ERR_H_SELECTED_UNIT_WRONG_VALUE : UINT := 901; (*Wrong value of selected hydraulic unit unit*)
	ERR_H_FIX_SPEED_IS_ZERO : UINT := 902; (*Fix pump speed is zero*)
	ERR_H_NO_DIR_CHANGE : UINT := 903; (*No change of pump move direction - check up and down sensors*)
	ERR_H_FILLING_TIME_LIMIT : UINT := 904; (*Filling - filling of A or B material is taking too long - check pressure sensors*)
	ERR_H_PUMP_SPEED_UP_TIME_LIMIT : UINT := 905; (*Speeding up pump is taking too long*)
	ERR_H_PUMP_REACH_PRES_TIME_LIMIT : UINT := 906; (*Reaching set pressure is taking too long*)
	ERR_H_NO_MATERIAL_WHILE_DOSSING : UINT := 907; (*During dosing system ran out of material*)
	ERR_H_FILL_CILI_NOT_DOWN_PRES_OK : UINT := 908; (*Filling pressure is reached, but hydraulic cilinder is not in down position*)
	ERR_H_PRESS_TOO_HIGH_A1 : UINT := 909; (*A1 component pressure is too high*)
	ERR_H_PRESS_TOO_HIGH_B1 : UINT := 910; (*B1 component pressure is too high*)
	ERR_H_PRESS_TOO_HIGH_A2 : UINT := 911; (*A2 component pressure is too high*)
	ERR_H_PRESS_TOO_HIGH_B2 : UINT := 912; (*B2 component pressure is too high*)
	ERR_H_PUMP_MOTOR_ERROR : UINT := 913; (*Hydraulic pump servo is in error*)
	ERR_MAT_EN_EX_IN_GLASS : UINT := 914; (*Material in mixer is too long - Make Cleaning or Dossing*)
END_VAR
(*Class 2 - warning*)
VAR CONSTANT
	ERR_H_A_MAT_SILO_EMPTY : UINT := 1020; (*White material silo is empty*)
	ERR_H_B_MAT_SILO_EMPTY : UINT := 1021; (*White material silo is empty*)
	ERR_H_BYPAS_SPEED_ZERO : UINT := 1022; (*Wrong hydraulic calibration - some of speed is zero*)
	ERR_DELTA_MIX_PRESSURE_TOO_LOW : UINT := 1023;
	ERR_M_MAT_IN_MIXER_TIME_1ST_WARN : UINT := 1024; (*Material in mixer is to long - Make Cleaning or Dossing*)
	ERR_M_MACHINE_MIXING : UINT := 1025; (*Material in mixer is to long - Make Cleaning or Dossing*)
END_VAR
(**)
(*Sealing Alarm 100..199*)
(**)
VAR CONSTANT
	ALERT_AUT_GLASS_IN_MACHINE : UINT := 100; (*Automatic mode error - in machine is unexpected glass*)
	ALERT_VAC_ERROR : UINT := 101;
	ALERT_SPATULA_TOut_Small : UINT := 102;
	ALERT_SPATULA_TOut_Last_Edge : UINT := 103;
	ALERT_SPATULA_TOut_Release : UINT := 104;
	ALERT_SPATULA_TOut_BIG_PISTON : UINT := 105;
	ALERT_SEALING_IO_NOT_PARKED : UINT := 106;
	ALERT_SEALING_IO_NOT_HOME : UINT := 107;
	ALERT_PARK_GLASS_IN_EXIT_UNIT : UINT := 108;
	ALERT_PARK_GLASS_IN_ENTRY_UNIT : UINT := 109;
	ALERT_PARK_GLASS_IN_SEAL_UNIT : UINT := 110;
	ALERT_PARK_VACUUM_ERROR : UINT := 111;
	ALERT_ENTRY_BUFFER_EMPTY : UINT := 112;
	ALERT_ENTRY_BUFFER_FULL : UINT := 113;
	ALERT_FINGER_NOT_FORWARD : UINT := 114;
	ALERT_S_COR_FILL_HYD_NOT_RDY : UINT := 115;
	ALERT_FINGER_OUT_OF_RANGE : UINT := 116;
	ALERT_SEAL_FINGER_NOT_CALIBRATED : UINT := 117;
	ALERT_SEAL_TIME_MAX_FILLING_TIME : UINT := 118;
	ALERT_EXITS_NOT_GEAR_OUT : UINT := 119;
END_VAR
(**)
(**)
(*Entry 1 Alarm 200..249*)
VAR CONSTANT
	ALERT_ENT_T_1_THICKNESS : UINT := 200;
	ALERT_ENT_1_SCL_Z_PARAMWRONG : UINT := 201;
	ALERT_ENT_1_SCL_Z_ENCODER : UINT := 202;
	ALERT_ENTRY1_IO_NOT_PARKED : UINT := 203;
	ALERT_ENTRY1_IO_NOT_HOME : UINT := 204;
	ALERT_STOP_SENS_BLINKED : UINT := 205;
	ALERT_HEADY_Y_SENS_BLINKED : UINT := 206;
END_VAR
(*Entry 2 Alarm 250..299*)
VAR CONSTANT
	ALERT_ENT_T_2_HOMING_TIMEOUT : UINT := 250;
	ALERT_ENT_T_2_DRIVER_FAULT : UINT := 251;
	ALERT_ENT_2_SCL_Z_PARAMWRONG : UINT := 252;
	ALERT_ENT_2_SCL_Z_ENCODER : UINT := 253;
	ALERT_ENTRY2_IO_NOT_PARKED : UINT := 254;
	ALERT_ENTRY2_IO_NOT_HOME1 : UINT := 255;
END_VAR
(*Exit 1 Alarm 300..349*)
VAR CONSTANT
	ALERT_EX_T_1_HOMING_TIMEOUT : UINT := 300;
	ALERT_EX_T_1_DRIVER_FAULT : UINT := 301;
	ALERT_EX_1_SCL_Z_PARAMWRONG : UINT := 302;
	ALERT_EX_1_SCL_Z_ENCODER : UINT := 303;
	ALERT_EX_1_BRD_CPT_HOMING_TOut : UINT := 304;
	ALERT_EX_1_BRD_CPT_Y2_SERVO : UINT := 305;
	ALERT_EX_1_BRD_CPT_NOT_DETECT : UINT := 306;
	ALERT_EX_1_BRD_CPT_SENSOR : UINT := 307;
	ALERT_EX_1_BRD_CPT_FB_ERROR : UINT := 308;
	ALERT_PARK_BRIGDE_1_SENS_ERR : UINT := 309;
	ALERT_EXIT1_IO_NOT_PARKED : UINT := 310;
	ALERT_EXIT1_IO_NOT_HOME : UINT := 311;
	ALERT_EXIT1_ENTRY_SENS_BLINKED : UINT := 312;
END_VAR
(*Exit 2 Alarm 350..399*)
VAR CONSTANT
	ALERT_EX_2_BRIDGE_HOMING_TIMEOUT : UINT := 350;
	ALERT_EX_2_BRIDGE_DRIVER_FAULT : UINT := 351;
	ALERT_EX_T_2_HOMING_TIMEOUT : UINT := 352;
	ALERT_EX_T_2_DRIVER_FAULT : UINT := 353;
	ALERT_EX_2_SCL_Z_PARAMWRONG : UINT := 354;
	ALERT_EX_2_SCL_Z_ENCODER : UINT := 355;
	ALERT_EX_2_SCL_BRDGE_PARAMWRONG : UINT := 356;
	ALERT_EX_2_SCL_BRDGE_ENCODER : UINT := 357;
	ALERT_EXIT2_IO_NOT_PARKED : UINT := 358;
	ALERT_EXIT2_IO_NOT_HOME : UINT := 359;
END_VAR
(*Exit 3 Alarm 400..449*)
VAR CONSTANT
	ALERT_EX_3_BRIDGE_HOMING_TIMEOUT : UINT := 400;
	ALERT_EX_3_BRIDGE_DRIVER_FAULT : UINT := 401;
	ALERT_EX_T_3_HOMING_TIMEOUT : UINT := 402;
	ALERT_EX_T_3_DRIVER_FAULT : UINT := 403;
	ALERT_EX_3_SCL_Z_PARAMWRONG : UINT := 404;
	ALERT_EX_3_SCL_Z_ENCODER : UINT := 405;
	ALERT_EX_3_SCL_BRDGE_PARAMWRONG : UINT := 406;
	ALERT_EX_3_SCL_BRDGE_ENCODER : UINT := 407;
	ALERT_EXIT3_IO_NOT_PARKED : UINT := 408;
	ALERT_EXIT3_IO_NOT_HOME : UINT := 409;
END_VAR
(*Exit 4 Alarm 450..499*)
VAR CONSTANT
	ALERT_EX_4_BRIDGE_HOMING_TIMEOUT : UINT := 450;
	ALERT_EX_4_BRIDGE_DRIVER_FAULT : UINT := 451;
	ALERT_EX_T_4_HOMING_TIMEOUT : UINT := 452;
	ALERT_EX_T_4_DRIVER_FAULT : UINT := 453;
	ALERT_EX_4_SCL_Z_PARAMWRONG : UINT := 454;
	ALERT_EX_4_SCL_Z_ENCODER : UINT := 455;
	ALERT_EX_4_SCL_BRDGE_PARAMWRONG : UINT := 456;
	ALERT_EX_4_SCL_BRDGE_ENCODER : UINT := 457;
	ALERT_EXIT4_IO_NOT_PARKED : UINT := 458;
	ALERT_EXIT4_IO_NOT_HOME : UINT := 459;
END_VAR
(**)
(*Entry 3 Alarm 500..549*)
VAR CONSTANT
	ALERT_ENT_T_3_HOMING_TIMEOUT : UINT := 500;
	ALERT_ENT_T_3_DRIVER_FAULT : UINT := 501;
	ALERT_ENT_3_SCL_Z_PARAMWRONG : UINT := 502;
	ALERT_ENT_3_SCL_Z_ENCODER : UINT := 503;
END_VAR
(*Entry 4 Alarm 550.599*)
VAR CONSTANT
	ALERT_ENT_T_4_HOMING_TIMEOUT : UINT := 550;
	ALERT_ENT_T_4_DRIVER_FAULT : UINT := 551;
	ALERT_ENT_4_SCL_Z_PARAMWRONG : UINT := 552;
	ALERT_ENT_4_SCL_Z_ENCODER : UINT := 553;
END_VAR
VAR
	New_Variable12 : UINT;
END_VAR
(*Exit 5 600..649*)
VAR CONSTANT
	ALERT_EX_T_5_HOMING_TIMEOUT : UINT := 600;
	ALERT_EX_T_5_DRIVER_FAULT : UINT := 601;
	ALERT_EX_5_SCL_Z_PARAMWRONG : UINT := 602;
	ALERT_EX_5_SCL_Z_ENCODER : UINT := 603;
	ALERT_EX_5_SCL_BRDGE_PARAMWRONG : UINT := 604;
	ALERT_EX_5_SCL_BRDGE_ENCODER : UINT := 605;
END_VAR
(*Exit 6 650..699*)
VAR CONSTANT
	ALERT_EX_T_6_HOMING_TIMEOUT : UINT := 650;
	ALERT_EX_T_6_DRIVER_FAULT : UINT := 651;
	ALERT_EX_6_SCL_Z_PARAMWRONG : UINT := 652;
	ALERT_EX_6_SCL_Z_ENCODER : UINT := 653;
	ALERT_EX_6_SCL_BRDGE_PARAMWRONG : UINT := 654;
	ALERT_EX_6_SCL_BRDGE_ENCODER : UINT := 655;
END_VAR
(*Exit 7 700..749*)
VAR CONSTANT
	ALERT_EX_T_7_HOMING_TIMEOUT : UINT := 700;
	ALERT_EX_T_7_DRIVER_FAULT : UINT := 701;
	ALERT_EX_7_SCL_Z_PARAMWRONG : UINT := 702;
	ALERT_EX_7_SCL_Z_ENCODER : UINT := 703;
	ALERT_EX_7_SCL_BRDGE_PARAMWRONG : UINT := 704;
	ALERT_EX_7_SCL_BRDGE_ENCODER : UINT := 705;
END_VAR
(*Exit 8 750..799*)
VAR CONSTANT
	ALERT_EX_T_8_HOMING_TIMEOUT : UINT := 750;
	ALERT_EX_T_8_DRIVER_FAULT : UINT := 751;
	ALERT_EX_8_SCL_Z_PARAMWRONG : UINT := 752;
	ALERT_EX_8_SCL_Z_ENCODER : UINT := 753;
	ALERT_EX_8_SCL_BRDGE_PARAMWRONG : UINT := 754;
	ALERT_EX_8_SCL_BRDGE_ENCODER : UINT := 755;
END_VAR
(*Info Alarmlar 1000...*)
VAR CONSTANT
	INFO_NOT_AUTO : UINT := 1000; (*Machine Not Auto*)
	INFO_EXIT2_HOMING_ERROR : UINT := 1001;
	INFO_EXIT3_HOMING_ERROR : UINT := 1002;
	INFO_EXIT4_HOMING_ERROR : UINT := 1003;
	INFO_CANNOT_MOVE : UINT := 1004;
	INFO_1_MaxDiffOver : UINT := 1005;
	INFO_2_MaxDiffOver : UINT := 1006;
	INFO_3_MaxDiffOver : UINT := 1007;
	INFO_4_MaxDiffOver : UINT := 1008;
END_VAR
(*ALERT_HOMING_GLASS_IN_MACHINE*)
(*Sealing Unit 100..199*)
(**** Max Single Alarm Constant*)
VAR CONSTANT
	MAX_SINGLE_ALARM_MIN1 : UINT := 1200; (**** Olabilecek maksimum single alarm sayisi*)
END_VAR
```

### GlobalAlert1.typ - Global data types
```iecst
(**)

TYPE
	gAlertType : 	STRUCT
		Abort : gAlertCommonType;
		Stop : gAlertCommonType;
		Pause : gAlertCommonType;
		Info : gAlertCommonType;
	END_STRUCT;
	gAlertCommonType : 	STRUCT
		Status : BOOL;
		IDX : ARRAY[0..MAX_SINGLE_ALARM_MIN1]OF BOOL;
	END_STRUCT;
END_TYPE

(**)
```

### Global.typ - Global data types
```iecst
TYPE
	gHMI_typ : 	STRUCT  (*Structure for handling visu*)
		IO_Control : gHMI_IO_Control_typ;
		UserName : STRING[80];
		Pulse : gHMIPulseType;
		Widget : gHMIWidgetType;
		MachineLock : gHMI_MachineLock_typ;
		CommUnit : gHMICommUnitType;
	END_STRUCT;
	gHMI_IO_Control_typ : 	STRUCT
		MaxForceValueLimit : UDINT; (*Maximum force value limit for I/O control page*)
		MinForceValueLimit : UDINT; (*Minimum force value limit for I/O control page*)
		SelectedSlotOld : USINT;
		SelectedSlot : USINT; (*Selected IO card slot*)
		FoceValue : ARRAY[0..15]OF UDINT; (*Force value for the IO channel*)
		ForceStatus : ARRAY[0..15]OF BOOL; (*Force status of the active IO card*)
		PhysicalStatus : ARRAY[0..15]OF UDINT; (*Physical value of the datapoint*)
		DatafieldStatus : ARRAY[0..15]OF BOOL; (*Controls the visibility of the datafields on the HMI*)
		BitmapSelector : USINT; (*Datapoin to select the picture to be shown on IO control page*)
		NameSelector : ARRAY[0..15]OF INT; (*IO Datapoint name selector for the active IO card*)
		MaxDpIndex : USINT; (*Number of chanels in curently selected card*)
		TypeOfIO : IOTypeChannel_enm; (*Type of card, that is currently used. DI DO AI AO*)
	END_STRUCT;
	gHMI_MachineLock_typ : 	STRUCT
		Logout : BOOL;
		Login : BOOL;
		Lock : BOOL;
		oldDay : USINT;
		EndTime : DATE_AND_TIME;
		Enable : BOOL;
		Password : STRING[80];
	END_STRUCT;
	gHMIWidgetType : 	STRUCT
		AlertLine : gHMIWidgetBtnGenType;
		AlertImage : gHMIWidgetBtnGenType;
		MachineLock : gHMIWidgetBtnGenType;
	END_STRUCT;
	gHMIPulseType : 	STRUCT
		ms50 : BOOL;
		ms100 : BOOL;
		ms200 : BOOL;
		ms300 : BOOL;
		ms500 : BOOL;
		ms1000 : BOOL;
	END_STRUCT;
	gHMIWidgetBtnGenType : 	STRUCT
		Enable : BOOL;
		Visible : BOOL;
		Style : STRING[20] := 'default';
		Image : STRING[80];
	END_STRUCT;
	gHMICommUnitType : 	STRUCT
		ActAlarms : UDINT;
	END_STRUCT;
END_TYPE
```

### Global1.var - Global variables
```iecst
VAR
	gIO : gIO_typ;
	gHMI : gHMI_typ;
	gAlert : gAlertType;
	FirstVariable : USINT;
END_VAR
(*HW Modules*)
VAR CONSTANT
	NUMBER_OF_MODULES : USINT := 12; (*Number of forceable I/O modules in the HW configuration*)
	NUMBER_OF_MODULES_MINUS_ONE : USINT := NUMBER_OF_MODULES-1; (*Number of forceable I/O modules in the HW configuration*)
	MAX_IO_MODULE_NUM : USINT := 14; (*Total number of IO modules currently in the machine*)
	MAX_IO_MODULE_NUM_MINUS_ONE : USINT := MAX_IO_MODULE_NUM-1; (*Total number of IO modules currently in the machine minus 1*)
END_VAR
(*
-----------------------------------------------------------------------------------------------------
IO Forcing
----------------------------------------------------------------------------------------------------*)
VAR CONSTANT
	NUMBER_OF_IO_MODULES : USINT := 17; (*Number of forceable I/O modules in the HW configuration*)
	NUMBER_OF_IO_MODULES_MINUS_1 : USINT := NUMBER_OF_IO_MODULES - 1; (*Number of forceable I/O modules in the HW configuration*)
	TOTAL_NUM_OF_ALL_MODULE : USINT := 17; (*Total number of modules currently in the machine (for chceking module status - X20 cards, IF modulex ...)*)
	TOTAL_NUM_OF_ALL_MODULE_MINUS_1 : USINT := TOTAL_NUM_OF_ALL_MODULE- 1; (*Total number of IO modules currently in the machine minus 1 (for chceking module status - X20 cards, IF modulex ...)*)
	IO_START_INDEX_SELECTED_SLOT : ARRAY[0..NUMBER_OF_IO_MODULES_MINUS_1] OF INT := [0,20,40,60,80,100,120,140,160,180,185,190,195,200,205,210,215]; (*Name of IO channel's start index in the text group "IO_Chanel_names"*)
	PI : REAL := 3.141593; (*Pi constant*) (*ERR_FUB_BUSY : UDINT := 65535; (*FUB busy*) (*ERR_OK : UDINT := 0; (*FUB executed successfully*)
END_VAR
(*Communication gMain*)
VAR
	gMain : gMain_typ;
	gCncAdress : UDINT;
END_VAR
```

### gMain.typ
```iecst
TYPE
	gMainOut_typ : 	STRUCT
		Status : gMainOutStatus_typ;
		MainStep : gMainState_Enum; (*Main step of main program*)
		MainSubStep : gMainSubState_Enum; (*Main sSUB step of main program*)
		Error : BOOL; (*Flag that machine has an active error*)
		ErrorCL0 : BOOL; (*Flag that critical error class 0 is active*)
		ErrorID : UDINT; (*Error ID of main logic*)
	END_STRUCT;
	gMain_typ : 	STRUCT
		In : gMainIn_typ;
		Out : gMainOut_typ;
	END_STRUCT;
	gMainOutStatus_typ : 	STRUCT  (*Main starus structure*)
		Active : BOOL;
		PoweredOn : BOOL; (*Flag to determine that machine axes are powered on*)
		Referenced : BOOL; (*Flag to determine that the machine is referenced*)
		ReadyToPowerOn : BOOL;
		MachineParked : BOOL; (*Flag that whole machine is in parking position*)
		StandStill : BOOL; (*Flag to determine that axes are standstill*)
		MoveActive : BOOL; (*Flag to signalize that some of axes is moving*)
		IO_Parked : BOOL; (*Flag that Inputs and Outputs of machine are in parking position*)
		Ax_Parked : BOOL; (*Flag to determine that Axes are in park (except X5 and X4)*)
		Ax_ParkedArray : ARRAY[0..MAX_AX_NR_MIN1]OF BOOL; (*Aray of flags showing whether is respective axis in parking pos. or not*)
		AxisDisabled : ARRAY[0..MAX_AX_NR_MIN1]OF BOOL; (*Flag that axis is disabled*)
		CurrentAutStep : UINT; (*Indication of actually executed automat Single step.*)
		AutoMode : BOOL; (*Flag that auto mode is active (standstill, running, stoped)*)
		CNC : gMainOutStatusCnc_typ;
	END_STRUCT;
	gMainOutStatusCnc_typ : 	STRUCT
		Active : BOOL;
	END_STRUCT;
	gMainIn_typ : 	STRUCT
		Enable : BOOL; (*Command to enable main control*)
		Cmd : gMainInCommands_typ; (*Main command structure*)
		Settings : gMainInSettings_typ; (*Main block settings*)
	END_STRUCT;
	gMainInCommands_typ : 	STRUCT  (*Main command structure*)
		Home : BOOL; (*Comand for starting the homing procedure*)
		Park : BOOL; (*Command for reaching the parking position*)
		Start : BOOL; (*Start command*)
		Stop : BOOL; (*Stop / pause commnad*)
		Load : BOOL; (*Command from pedal to start loading*)
		Reset : BOOL; (*Reset commnad*)
		SetMultiturnEncoder : BOOL; (*Set multiturn offset*)
		MultiturnEncHomeLimSwitch : BOOL; (*Home to limit switch*)
		MultiturnEncHomeOffsetValue : BOOL; (*Home to offset value*)
		Manual : ManualCommands_typ; (*Comands for manual movement*)
	END_STRUCT;
	ManualCommands_typ : 	STRUCT  (*Comands for manual movement*)
		InvJogPos : BOOL; (*Cmd to jog with asynchronous motor*)
		InvJogNeg : BOOL; (*Cmd to jog with asynchronous motor*)
		JogPos : ARRAY[0..MAX_AX_NR_MIN1]OF BOOL; (*Jog Negative commands*)
		JogNeg : ARRAY[0..MAX_AX_NR_MIN1]OF BOOL; (*Jog Positive commands*)
		GoToPos_Stop : BOOL; (*Cmd to go to selected position with axis or stop during movement*)
		SetPos : REAL; (*Position where to move selected axis*)
		ActiveAx : ARRAY[0..MAX_AX_NR_MIN1]OF BOOL; (*Indication which axis is selected in visu - identical indexes with main program*)
	END_STRUCT;
	gMainInSettings_typ : 	STRUCT  (*Main block settings*)
		SelectedMode : USINT; (*Represents the selected operation mode, 0 Manual; 1 - automatic single step mode; 2 continous Automat*)
		AxisSelected : ARRAY[0..MAX_AX_NR_MIN1]OF BOOL; (*Enable or disable axis (0 - Axis disabled, 1 - Axis enabled)*)
		ParkPos : ARRAY[0..MAX_AX_NR_MIN1]OF REAL; (*Parking positions for axes*)
		ParPosZaxis : REAL; (*Parking position of Z axis [units]*)
		MultiEncSettings : gMainInSettingsMultiEnc_typ; (*Structure with parameters for settings multiturn encoders*)
	END_STRUCT;
	gMainInSettingsMultiEnc_typ : 	STRUCT
		reserved : USINT;
	END_STRUCT;
	gMainState_Enum :
		(
		MAIN_INIT := 0,
		MAIN_WAIT_CMD,
		MAIN_MANUAL_MOVE,
		MAIN_START,
		MAIN_STOP,
		MAIN_PAUSE,
		MAIN_PARK,
		MAIN_HOME,
		MAIN_RESET,
		MAIN_NEW_LAYOUT,
		MAIN_AUTO_STANDSTILL,
		MAIN_AUTO_RUNNING,
		MAIN_AUTO_STOPPED,
		MAIN_MULTI_ENCODER_OFFSET,
		MAIN_HOME_LIMIT_SWITCH,
		MAIN_GO_SET_ORIJIN,
		MAIN_AUTO_DETECT_ORIGIN,
		MAIN_TRANSFER_TO_BT,
		MAIN_TRANSFER_FROM_LD,
		MAIN_GET_ENC_OFFSET_AXIS_B,
		MAIN_ERROR
		);
	gMainSubState_Enum :
		(
		SUB_INIT,
		SUB_CHECK_IO,
		SUB_HOME_START,
		SUB_PARK_START,
		SUB_CMD_DONE,
		SUB_STOP,
		SUB_ERROR
		);
END_TYPE
```

### GlobalIO.typ
```iecst
TYPE
	gIO_BreakerOut_typ : 	STRUCT
		FanDoorControl : BOOL;
		FanStart : BOOL;
		WorkEnable : BOOL;
		TableValveUpSlow : BOOL;
		TableValveDownSlow : BOOL;
		TableDownValve : BOOL;
		TableUpValve : BOOL;
		HydraulicPumpStart : BOOL;
		PositionersUpValve : BOOL;
		PositionersDownValve : BOOL;
		LeftCarrierUp : BOOL;
	END_STRUCT;
	gIO_BreakerIn_typ : 	STRUCT
		BT_EStop : BOOL; (* BT = Breaker Table *)
		BT_IsUpSW : BOOL; (* BT = Breaker Table *)
		BT_IsUpSlowSW : BOOL; (* BT = Breaker Table *)
		BT_IsDownSW : BOOL; (* BT = Breaker Table *)
		BT_IsDownSlowSW : BOOL; (* BT = Breaker Table *)
		BT_TransferBtn : BOOL; (* BT = Breaker Table *)
		BT_FanStartPedal : BOOL; (* BT = Breaker Table *)
		BT_FanMotorFault : BOOL; (* BT = Breaker Table *) (* Axis*)
		BT_CarrierIsUpSW : USINT; (* BT = Breaker Table *)
		BT_HydPumpMotorFault : USINT; (* BT = Breaker Table *)
	END_STRUCT;
	gIO_InCT_typ : 	STRUCT  (*Cutting Table Input Types*)
		EmergencyStop : BOOL; (*Emergency Stop Input to make an emergency stop*)
		PhaseRelayFault : BOOL; (*Phase Relay Fault detection*)
		ResetButton : BOOL; (*Reset Button to reset any faults*)
		StartButton : BOOL; (*Start button to start machine in automade*)
		PauseButton : BOOL; (*Pause button to pause the machine during cut*)
		FanMotorFault : BOOL; (*Fan Motor Fault detection for cutting table and breaker table*)
		SetPressureReached : BOOL; (*Cutting pressure reached set value, feedback signal*)
		FanPedal : BOOL; (*Manual Pedal control input for table fan start (toggle input)*)
		LowAirPressure : BOOL; (*Low air pressure sensor*) (* ockm*)
		TableDownSlowSwicth : BOOL; (*OCKM*)
		TableUpSlowSwicth : BOOL; (*OCKM*)
		TableUpStopSwicth : BOOL; (*OCKM*)
		TableDownStopSwicth : BOOL; (*OCKM*)
		HydraulicMotorTermic : BOOL; (*OCKM*)
		HydraulicMotorRun : BOOL; (*OCKM*)
		GlassSearchSensor : BOOL;
		HeadMaxDownSensor : BOOL;
		TableSquareBack : BOOL; (*FCL*)
		GlassTransBeltIsDown : BOOL; (*FCL*)
		GlassStopSW : BOOL; (*FCL*)
		GlassExitSW : BOOL; (*FCL*)
		AxisX_PositiveLimit : BOOL;
		AxisX_NeativeLimit : BOOL;
		AxisX_ReferenceLimit : BOOL; (*AX_X*)
		AxisY_ReferenceLimit : BOOL; (*AX_Y*)
		AxisC_ReferenceLimit : BOOL; (*AX_C*)
	END_STRUCT;
	gIO_In_typ : 	STRUCT
		Breaker : gIO_BreakerIn_typ;
		CT : gIO_InCT_typ; (*CT = Cutting Table*)
		Loader : gIO_Out_Loader_typ;
	END_STRUCT;
	gIO_Out_CT_typ : 	STRUCT
		RedLamp : BOOL; (*Red Lamp On if Error Occured*)
		YellowLamp : BOOL; (*Yellow Lamp On if manual activation *)
		GreenLamp : BOOL; (*Green Lamp On if machine cutting*)
		Reset : BOOL; (*Reset output signal*)
		CuttingHeadDown : BOOL; (*Send Cutting Head Down to glass surface*)
		DiamondOil : BOOL; (*Oil SupplyTANK Selection Tank-2*)
		LowEMotorStart : BOOL; (*Start LowE Motor  , Start and Stop conttroled by one output*)
		LowEMotorDown : BOOL; (*Low_e Motor UP and Down Controlled by one output*)
		FanDoorClose : BOOL; (*Close door in fan for blowers*)
		FanStart : BOOL; (*Table Fan Start Command*)
		SquareForward : BOOL; (*Move forward square system*) (* OCKM*)
		HydraulicMotorStart : BOOL;
		TableUpValve : BOOL; (*OCKM*)
		TableDownValve : BOOL; (*OCKM*)
		TableUpSlowValve : BOOL; (*OCKM*)
		TableDownSlowValve : BOOL; (*OCKM*)
		SquareUpValve : BOOL; (*OCKM*)
		SquareDownValve : BOOL; (*OCKM*)
		XYGlassBreakControl : BOOL; (*OCKM*)
		TransferBelt : BOOL;
		AO_CuttingPressure : USINT; (*Analog Output Cutting Pressure*)
	END_STRUCT;
	gIO_Out_Loader_typ : 	STRUCT
		New_Member : USINT;
	END_STRUCT;
	gIO_Out_typ : 	STRUCT
		CT : gIO_Out_CT_typ;
		Breaker : gIO_BreakerOut_typ;
		Loader : gIO_Out_Loader_typ;
	END_STRUCT;
	gIO_typ : 	STRUCT
		In : gIO_In_typ;
		Out : gIO_Out_typ;
	END_STRUCT;
END_TYPE
```

### Parameters.typ - Global data types
```iecst
(********************************************************************
 * COPYRIGHT -- Bernecker + Rainer
 ********************************************************************
 * Package: CuttingTable
 * File: Parameter.typ
 * Author: blanca-gutim
 * Created: December 07, 2012
 ********************************************************************
 * Data types of package CuttingTable
 ********************************************************************)
(**)
(*========================================================================================================*)
(*Structure with machine parameters*)
(*========================================================================================================*)

TYPE
	gMachineType_Enum :
		(
		FCM := 0,
		FCL := 1,
		OCKM := 2,
		YCKM := 3,
		YCKM_BREAKER := 4
		);
	gParameters_type : 	STRUCT
		BridgeStraight : BOOL; (*Command is taken from the HMI when the bridge straightness is set by the user*)
		MachineType : gMachineType_Enum; (*Machine type  FCM= 0 FCL= 1 OCKM= 2 YCKM =3 YCKM_BREAKER = 4*)
		Options : Parameters_Options_typ;
		LengthParametes : LengthParametes_type; (*Length parameters*)
		DriverParameters : ARRAY[0..5]OF DriverParameters_type; (*Drive parameters*)
		PressParameters : PressParameters_type; (*Pressure parameters*) (*		LoaderParameters : LoaderCtrl_In_Par_typ; (*Loader parameters*)
		Network : Recipe_Ctrl_In_Par_Net_typ; (*Network parameters*)
	END_STRUCT;
END_TYPE

(**)
(*========================================================================================================*)
(*Options*)
(*========================================================================================================*)

TYPE
	Parameters_Options_typ : 	STRUCT
		HW : Parameters_Options_HW_typ; (*Cutting table HW options*)
		SW : Parameters_Options_SW_typ; (*Cutting table SW options*)
	END_STRUCT;
	Parameters_Options_HW_Gantry_typ : 	STRUCT
		Active : BOOL;
		HoldingBrakes : BOOL;
		MultiturnEnc : BOOL;
	END_STRUCT;
	Parameters_Options_HW_typ : 	STRUCT
		LinearMotors_v1 : BOOL;
		LinearMotors_v2 : BOOL;
		NewLowE : BOOL; (*New version of the Low-E*)
		InkJet : {REDUND_UNREPLICABLE} BOOL; (*Inkjet printer exists in the machine instead of the old labeler system*)
		Labeler : BOOL;
		CAxisRev0 : BOOL; (*Revision xx-0 for the C axis [since it's a resolver, this should be known within the system so that the HW cfg is done accordingly]*)
		Gantry : Parameters_Options_HW_Gantry_typ;
		OCKMEnableTransferToBT : BOOL; (*Requested by the customer for one machine [14.05.2015].
The feature enables the glass transfer from the table to another machine in line. The process is the same with the YCKM_BREAKERs*)
	END_STRUCT;
	Parameters_Options_SW_typ : 	STRUCT
		TorqueDiffTimeout : REAL;
		TorqueDiffLimit : REAL;
		GanTorqMonTimeoutError : USINT; (*Option to treat the torque difference monitoring timeout as an error; by default it is treated as a warning*)
		NewGCodeRecipe : BOOL;
		GantryTorqueMonActive : BOOL; (*Option to activate the torque difference monitoring *)
		KeepBridgeEnabled : BOOL; (*Option keep the bridge axes enabled all the time*)
		AutoHwCfg : BOOL;
		AutoUserLogout : BOOL; (*Option to de/activate the automatic user logout functionality*)
		ManualOptimization : BOOL; (*Option to de/activate the manual optimization feature (since version  A3.54.0)*)
		LanguageEnable : ARRAY[0..9]OF BOOL; (*Enable the corresponding language to make it selectible on the HMI when the translations are there*)
	END_STRUCT;
END_TYPE

(**)
(*========================================================================================================*)
(*Length parameters*)
(*========================================================================================================*)

TYPE
	LengthParametes_type : 	STRUCT
		BAxisHomePos : REAL;
		BAxisMultiSetPos : REAL;
		YAxisMultiSetPos : REAL; (*Multiturn encoder home offset value for the Y axis [mm] / 0 when not applicable*)
		YAxisMultiHomeOffset : REAL; (*Set position for the multiturn encoder for the Y axis [mm] / 0 when not applicable*)
		MasterHomeOffset : REAL; (*Multiturn encder home offset value for master X axis [mm]*)
		MasterMultiSetPos : REAL; (*Set position of the multiturn encoder for the master*)
		SlaveHomeOffset : REAL; (*Multiturn encder home offset value for slave X2 axis [units]*)
		SlaveMultiSetPos : REAL; (*Set position of the multiturn encoder for the slave*)
		HeadUpTime : REAL; (*Time for the cutting head to move up [s]*)
		HeadDownTime : REAL; (*Time for the cutting head to move down [s]*)
		Low_eAboveTime : REAL; (*Time for the Low-E head to move up [s]*)
		Low_eBelowTime : REAL; (*Time for the Low-E head to move down [s]*)
		WaitPressureTime : REAL; (*Time to wait for the pressure reached [s]*)
		SquareForwardTime : REAL; (*Time to wait for the square forward movement [s]*)
		StretchingTime : REAL; (*Time to define how long the oil must be pumped when the machine starts operation [s] - NOT USED NOW*)
		X_GlassOriginPos : REAL; (*X distance between the Reference position and the Glass Origin position when the glass is placed without shift or rotation [mm]*)
		Y_GlassOriginPos : REAL; (*Y distance between the Reference position and the Glass Origin position when the glass is placed without shift or rotation [mm]*)
		C_GlassOriginPos : REAL; (*Offset between the cutting head and the glass (alignment) [°] - IT HAS TO BE MEASURED*)
		Y_GlassOriginPos_Right : REAL; (*Y distance between the Glass Origin position in the right side of the machine and the positive software limit in Y direction[mm] - ONLY IN FCL BIG SIZE MACHINES*)
		OffsetSpeed : REAL; (*Speed to move to Origin position [% prespect to maximum speed]*)
		X_AxisOffsetMachine : REAL; (*X offset between the cutting head and the laser sensor [mm]*)
		Y_AxisOffsetMachine : REAL; (*Y offset between the cutting head and the laser sensor [mm]*)
		Distance_Lowe_CuttingHead_X : REAL; (*X distance between cutting head and Low-E head [mm] *)
		Distance_Lowe_CuttingHead_Y : REAL; (*Y distance between cutting head and Low-E head [mm]*)
		X_HomeOffsetPos : REAL; (*X axis home offset [mm] - IT DEFINES THE REFERENCE POSITION, WHERE AXES ARE 0 units*)
		Y_HomeOffsetPos : REAL; (*Y axis home offset [mm] - IT DEFINES THE REFERENCE POSITION, WHERE AXES ARE 0 units*)
		C_HomeOffsetPos : REAL; (*C axis home offset [°] - IT DEFINES THE REFERENCE POSITION, WHERE AXES ARE 0 units*)
		ParkSpeed : REAL; (*Speed to move to Park position [% prespect to maximum speed]*)
		X3_Offset : REAL;
		X2_Offset : REAL;
		Y1_Offset : REAL;
		X_SafeLoadPosition : REAL; (*X axis position mandatory before loading*)
		MoveSafeLoadSpeed : REAL; (*Speed at which bridge will move to safe loading position*)
		Y_SafeLoadPosition : REAL; (*Y axis position mandatory before loading*)
		X_GlassTransferEndPosition : REAL; (*X axis, end position of transfer of the glass to breaking table*)
		Y_GlassTransferEndPosition : REAL; (*Y axis, end position of transfer of the glass to breaking table*)
		HomeSpeedTrigger : REAL;
		AutoSquaringSpeed : REAL; (*Auto squaring speed from the memory*)
		PushGlassSpeed : REAL; (*Speed at which glass should be transfered pushed after loading*)
		TransferSpeed : REAL; (*Speed at which glass should be transfered to breaking table*)
		StraightBridgeDelta : DINT; (*Defined by user, offset between ref pulses of X and X2 axes, having this parameter we can establish straigh position of bridge*)
		X_PushPositionEnd : REAL; (*Position when to finish glass pushing*)
		Y_PushPositionEnd : REAL; (*Position when to finish glass pushing*)
		Y_TransferPositionStart : REAL; (*Position when to start glass pushing/transfering*)
		X_TransferPositionStart : REAL; (*Position when to start glass pushing/transfering*)
		LabelApplyTime : REAL; (*Label application time*)
		InkJetPrintStroke : {REDUND_UNREPLICABLE} REAL; (*Stroke within which the inkjet should print*)
		InkJetPrintSpeed : {REDUND_UNREPLICABLE} REAL; (*Optimum speed at which the inkjet should perform the print (PLC will check the actual path speed of the CNC and trigger the print)*)
	END_STRUCT;
END_TYPE

(*========================================================================================================*)
(*Drive parameters*)
(*========================================================================================================*)

TYPE
	DriverParameters_type : 	STRUCT
		Enabled : BOOL;
		CntDir : USINT; (*Encoder counting direction*)
		DriveStep : REAL; (*Units needed for the motor to complete one turn [um] - THE SAME THAN units IN LOAD IN ACP INIT TABLE*)
		PositiveLimit : REAL; (*Positive software limit [mm] - THE SAME THAN IN LOAD IN ACP INIT TABLE*)
		NegativeLimit : REAL; (*Negative software limit [mm] - THE SAME THAN IN LOAD IN ACP INIT TABLE*)
		PID : DriverParameters_PID_type; (*PID parameters - THE SAME THAN IN CONTROLLER IN ACP INIT TABLE*)
	END_STRUCT;
END_TYPE

(*========================================================================================================*)
(*Drive PID parameters*)
(*========================================================================================================*)

TYPE
	DriverParameters_PID_type : 	STRUCT
		A0 : REAL;
		A1 : REAL;
		B0 : REAL;
		B1 : REAL;
		FilterType : UINT;
		Mode : USINT; (*Controller mode*)
		SpeedController : DriverParameters_PID_kv_tn_type; (*PID parameters for speed controller*)
		PositionController : DriverParameters_PID_kv_tn_type; (*PID parameters for position controller*)
		FeedForward : DriverParameters_FF_type; (*Feed forward related parameters*)
	END_STRUCT;
END_TYPE

(*========================================================================================================*)
(*Drive PID parameters: kn and tv*)
(*========================================================================================================*)

TYPE
	DriverParameters_PID_kv_tn_type : 	STRUCT
		kv : REAL; (*Proportional amplification*)
		tn : REAL; (*Integral action time [s]*)
	END_STRUCT;
END_TYPE

(*========================================================================================================*)
(*Drive Feed forward parameters*)
(*========================================================================================================*)

TYPE
	DriverParameters_FF_type : 	STRUCT
		Torque_Pos : REAL; (*Torque in positive direction [Nm]*)
		Torque_Neg : REAL; (*Torque in negative direction [Nm]*)
		Torque_Load : REAL; (*Load torque [Nm]*)
		Kv_Torque : REAL; (*Speed torque factor [Nms]*)
		Inertia : REAL; (*Mass moment of inertia [kgm˛]*)
	END_STRUCT;
END_TYPE

(*========================================================================================================*)
(*Pressure parameters*)
(*========================================================================================================*)

TYPE
	PressParameters_type : 	STRUCT
		PressureCalibration : REAL; (*Coefficient to convert pressure value in Analog Output*)
		PressureCoefficent : REAL; (*Indicates the pressure value set in Automatic Mode page*)
		HeadDownPress : REAL; (*Pressure when the cutting head is moving down [bar]*)
		VinylCutPressure : REAL; (*Pressure when the vynil cutting is done*)
		LoweDownPressure : REAL; (*Low-e down pressure - used only for the new low-e system *)
		GlassType : Press_Params_Glass_type; (*Parameters dependent on the glass type*)
	END_STRUCT;
END_TYPE

(*========================================================================================================*)
(*Pressure parameters that are dependent on the glass type*)
(*========================================================================================================*)

TYPE
	Press_Params_Glass_type : 	STRUCT
		T2 : Glass_PressureType; (*Glass thickness equal to 2 mm*)
		T3 : Glass_PressureType; (*Glass thickness equal to 3 mm*)
		T4 : Glass_PressureType; (*Glass thickness equal to 4 mm*)
		T5 : Glass_PressureType; (*Glass thickness equal to 5 mm*)
		T6 : Glass_PressureType; (*Glass thickness equal to 6 mm*)
		T8 : Glass_PressureType; (*Glass thickness equal to 8 mm*)
		T10 : Glass_PressureType; (*Glass thickness equal to 10 mm*)
		T12 : Glass_PressureType; (*Glass thickness equal to 12 mm*)
		T15 : Glass_PressureType; (*Glass thickness equal to 15 mm*)
		T19 : Glass_PressureType; (*Glass thickness equal to 19 mm*)
	END_STRUCT;
END_TYPE

(*========================================================================================================*)
(*Pressure parameters that are dependent on the glass type*)
(*========================================================================================================*)

TYPE
	Glass_PressureType : 	STRUCT
		MFunctionStart : UINT; (*Value of the fist M-Function used for this pressure values*)
		Pressure : ARRAY[0..5]OF REAL; (*Set pressure for different kinds of cut [bar]*)
	END_STRUCT;
END_TYPE
```

### Parameters.var - Global variables
```iecst
(********************************************************************
 * COPYRIGHT -- Bernecker + Rainer
 ********************************************************************
 * Package: MachineManager
 * File: MachineManager.var
 * Author: blanca-gutim
 * Created: December 04, 2012
 ********************************************************************
 * Variables of package MachineManager
 ********************************************************************)
(**)
(*
VAR CONSTANT
	FCM : USINT := 0;
	FCL : USINT := 1;
	OCKM : USINT := 2;
	YCKM : USINT := 3;
	YCKM_BREAKER : USINT := 4;
END_VAR
*)
(*========================================================================================================*)
(*Cutting table parameters structure*)
(*========================================================================================================*)
VAR RETAIN
	gOldOffset : REAL := 0.0; (*Previous homing offset for th C axis*)
	gParameters : gParameters_type; (*Cutting table parametesr structure*)
	gTotalCounter : UDINT; (*Total counter variable*)
	gDailyCounter : UDINT; (*Daily counter variable*)
	gSpeedRate : REAL; (*Speed rate variable*)
	gPressureRate : REAL; (*Pressure variable*)
	gDay : DATE; (*Variable with day information*)
	gMaxWorkCycles : UDINT; (*Maximum number of cycles until the machine is locked*)
END_VAR
VAR
	gFactorySettings : gParameters_type; (*Structure with the factory settings*)
END_VAR
```

### Motion.var
```iecst
VAR
	gAxBasic : ARRAY[0..MAX_AX_NR_MIN1] OF MpAxisBasic;
	gAxBasicPar : ARRAY[0..MAX_AX_NR_MIN1] OF MpAxisBasicParType;
END_VAR
VAR CONSTANT
	C_MAX_CUT_SPEED : REAL := 200.0; (*Maximum speed of the path while cutting [m/min]*)
	C_MAX_C_AXIS_SPEED : REAL := 1440.0; (*Maximum speed of the C axis [°/s]*)
	AX_X : USINT := 0;
	AX_Y : USINT := 1;
	AX_C : USINT := 2;
	AX_B : USINT := 3;
	AX_VC : USINT := 4;
	MAX_AX_NR_MIN1 : USINT := 5;
END_VAR
```

- Project.language (not shown)

### Program Logical/SourceCode/MAIN (IEC)

#### Cyclic.st - Cyclic code
```iecst
PROGRAM _CYCLIC
	IF gCncAdress > 0 THEN
		pCNC ACCESS gCncAdress;
	ELSE
		RETURN;
	END_IF;

	fbCuttingTransfer_0();

	fbTableUpDown_0();

	AxesStatus;

	CASE gMain.Out.MainStep OF

		MAIN_INIT:

			IF Loc.FirstInMainState THEN
				gMain.Out.MainSubStep := SUB_INIT;
			ELSE
				;
			END_IF;

		MAIN_WAIT_CMD:
		MAIN_MANUAL_MOVE:
		MAIN_START:
		MAIN_STOP:
		MAIN_PAUSE:
		MAIN_PARK:
		MAIN_HOME:
		MAIN_RESET:
		MAIN_NEW_LAYOUT:
		MAIN_AUTO_STANDSTILL:
		MAIN_AUTO_RUNNING:
		MAIN_AUTO_STOPPED:
		MAIN_MULTI_ENCODER_OFFSET:
		MAIN_HOME_LIMIT_SWITCH:
		MAIN_GO_SET_ORIJIN:
		MAIN_AUTO_DETECT_ORIGIN:
		MAIN_TRANSFER_TO_BT:
		MAIN_TRANSFER_FROM_LD:
		MAIN_GET_ENC_OFFSET_AXIS_B:
		MAIN_ERROR:

	END_CASE;

	Loc.FirstInMainState := gMain.Out.MainStep <> Loc.OldMainState;
	Loc.OldMainState	 := gMain.Out.MainStep;

	Loc.FirstInSubState	:= gMain.Out.MainSubStep <> Loc.OldSubState;
	Loc.OldSubState 	:= gMain.Out.MainSubStep;

END_PROGRAM
```

#### Init.st - Init code
```iecst
PROGRAM _INIT

END_PROGRAM
```

#### Types.typ - Local data types
```iecst
TYPE
	Timers_typ : 	STRUCT
		TON_HomeState : TON;
		TON_ParkState : TON;
	END_STRUCT;
	Loc_typ : 	STRUCT
		FirstInSubState : BOOL;
		FirstInMainState : BOOL;
		OldSubState : gMainSubState_Enum;
		OldMainState : gMainState_Enum;
		Timers : Timers_typ;
	END_STRUCT;
END_TYPE
```

#### Variables.var - Local variables
```iecst
VAR
	fbCuttingTransfer_0 : fbCuttingTransfer;
	EnabledFlag : BOOL;
	PowerFlag : BOOL;
	ReferencedFlag : BOOL;
	StandStillFlag : BOOL;
	MoveActiveFlag : BOOL;
	DrivesReadyFlag : BOOL; (*DrivesAreReadyToPowerOn*)
	i : USINT;
	pCNC : REFERENCE TO MpCnc3Axis;
	Loc : Loc_typ;
	fbTableUpDown_0 : fbTableUpDown;
END_VAR
```

#### AxesStatus.st
```iecst
ACTION AxesStatus:

	//------------------
	// Checks all Axes are enabled or not
	EnabledFlag := TRUE;
	FOR i := 0 TO MAX_AX_NR_MIN1 DO
		IF NOT  gAxBasic[i].Active AND gParameters.DriverParameters[i].Enabled  THEN
			EnabledFlag := FALSE;
			EXIT;
		END_IF;
	END_FOR;
	//------------------

	//------------------
	// Checks all Axes are powered or not
	PowerFlag := TRUE;
	FOR i := 0 TO MAX_AX_NR_MIN1 DO

		IF NOT  gAxBasic[i].PowerOn AND gParameters.DriverParameters[i].Enabled THEN
			PowerFlag := FALSE;
			EXIT;
		END_IF;

	END_FOR;
	//------------------

	//------------------
	// Checks all Axes are referenced or not
	ReferencedFlag := TRUE;
	FOR i := 0 TO MAX_AX_NR_MIN1 DO

		IF NOT  gAxBasic[i].IsHomed AND gParameters.DriverParameters[i].Enabled  THEN
			ReferencedFlag := FALSE;
			EXIT;
		END_IF;

	END_FOR;

	//--------------
	// Drive Ready Flag
	DrivesReadyFlag   := TRUE;
	FOR i := 0 TO MAX_AX_NR_MIN1 DO
		IF NOT  gAxBasic[i].Info.ReadyToPowerOn  AND gParameters.DriverParameters[i].Enabled THEN
			DrivesReadyFlag := FALSE;
			EXIT;
		END_IF;
	END_FOR;

	// ----------------------------------------
	//Standstill
	// ----------------------------------------
	StandStillFlag := TRUE;
	FOR i := 0 TO MAX_AX_NR_MIN1 BY 1 DO
		IF  NOT (gAxBasic[i].Info.AxisAdditionalInfo.PLCopenState = mcAXIS_STANDSTILL) AND  gParameters.DriverParameters[i].Enabled THEN
			StandStillFlag := FALSE;
			EXIT;
		END_IF
	END_FOR

	// ----------------------------------------
	//MoveActive
	// ----------------------------------------
	MoveActiveFlag := TRUE;
	FOR i := 0 TO MAX_AX_NR_MIN1 BY 1 DO
		IF  (gAxBasic[i].MoveActive) AND  gParameters.DriverParameters[i].Enabled THEN
			MoveActiveFlag := FALSE;
			EXIT;
		END_IF
	END_FOR

	// ----------------------------------------
	//Park Pos Control
	// ----------------------------------------
	IF  (ABS(gMain.In.Settings.ParkPos[AX_X] - gAxBasic[AX_X].Position)<= 5.0 ) AND
		(ABS(gMain.In.Settings.ParkPos[AX_Y] - gAxBasic[AX_Y].Position)<= 5.0 ) THEN
		gMain.Out.Status.Ax_Parked := TRUE;
	ELSE
		gMain.Out.Status.Ax_Parked := FALSE;
	END_IF;

	gMain.Out.Status.Active				:= EnabledFlag;

	gMain.Out.Status.PoweredOn 			:= PowerFlag;

	gMain.Out.Status.Referenced 		:= ReferencedFlag;

	gMain.Out.Status.ReadyToPowerOn 	:= DrivesReadyFlag;

	gMain.Out.Status.StandStill 		:= StandStillFlag;

	gMain.Out.Status.MoveActive 		:= MoveActiveFlag;

	gMain.Out.Status.CNC.Active			:= pCNC.Active;

END_ACTION
```

#### Reference.st
```iecst
ACTION Reference:

	IF gMain.Out.Error THEN
		gMain.Out.MainSubStep			:= SUB_ERROR;
	END_IF

	CASE gMain.Out.MainSubStep  OF

		SUB_INIT:

			IF Loc.FirstInHomeState THEN
				gIO.Out.CT.CuttingHeadDown 		:= FALSE;
				gIO.Out.CT.LowEMotorDown   		:= FALSE;
				gIO.Out.CT.FanStart		   		:= FALSE;
				gIO.Out.CT.XYGlassBreakControl  := FALSE;
				gIO.Out.CT.TransferBelt			:= FALSE;
				gIO.Out.CT.SquareForward		:= FALSE;
				Loc.Timers.TON_HomeState.IN		:= FALSE;
				gAxBasic[AX_X].Home				:= FALSE;
				gAxBasic[AX_Y].Home				:= FALSE;
				gAxBasic[AX_C].Home				:= FALSE;
			ELSE

				Loc.Timers.TON_HomeState.IN := TRUE;
				Loc.Timers.TON_HomeState.PT := T#1s;
				IF Loc.Timers.TON_HomeState.Q THEN
					Loc.Timers.TON_HomeState.IN := FALSE;
					Loc.HomeState			:= HOME_CHECK_IO;
				END_IF

			END_IF;

		SUB_CHECK_IO:

			IF NOT gIO.In.CT.HeadMaxDownSensor THEN
				gMain.Out.Error 	:= TRUE;
				gMain.Out.ErrorID 	:= 999; // Diamond Is Not Back
				gMain.Out.MainSubStep   	:= SUB_ERROR;
				RETURN;

			ELSIF gParameters.MachineType = OCKM THEN
				IF NOT gIO.In.CT.TableDownStopSwicth OR gIO.In.CT.TableUpSlowSwicth ELSE
					gMain.Out.Error 	:= TRUE;
					gMain.Out.ErrorID 	:= 999; // CT_Is_Not_Down
					gMain.Out.MainSubStep   	:= SUB_ERROR;
					RETURN;
				ELSIF NOT gIO.In.CT.TableSquareBack THEN
					gMain.Out.Error 	:= TRUE;
					gMain.Out.ErrorID 	:= 999; // CT_Is_Squares_Are_Not_Back
					gMain.Out.MainSubStep   	:= SUB_ERROR;
					RETURN;
				ELSE
				;
				END_IF // OCKM
			ELSIF gParameters.MachineType = FCL THEN
				IF NOT gIO.In.CT.GlassTransBeltIsDown ELSE
					gMain.Out.Error 	:= TRUE;
					gMain.Out.ErrorID 	:= 999; // CT_Belt Is Not Down
					gMain.Out.MainSubStep   	:= SUB_ERROR;
					RETURN;
				END_IF // FCL
			ELSE
					// Home Start
					gMain.Out.MainSubStep   	:= SUB_HOME_START;

			END_IF;

		SUB_HOME_START:

				IF Loc.FirstInSubState THEN
					gAxBasicPar[AX_X].Homing.Mode					:= mcHOMING_ABSOLUTE_SWITCH;
					gAxBasicPar[AX_X].Homing.Options.SensorOffset   := gParameters.LengthParametes.X_HomeOffsetPos; //gFixData.Ax[AX_X].Config.MultiturnEncOffset; //Home yaptiktan sonra kaçinci pozisyona kadar gitsin
					gAxBasicPar[AX_X].Homing.Position 			  	:= 0; /gFixData.Ax[AX_X].Par.Homing.Position; //Home yapip Sensor offset kadar gidip bunuda üstüne ekliyor
					gAxBasicPar[AX_X].Homing.Options.SwitchEdge     := mcDIR_NEGATIVE; //Switch nerede aranacak
					gAxBasicPar[AX_X].Homing.Options.HomingDirection:= mcDIR_POSITIVE; //switch ten kurtulduktan sonra offset için hangi yöne gidecek
					gAxBasicPar[AX_X].Homing.Options.StartDirection := mcDIR_NEGATIVE;
					gAxBasicPar[AX_X].Homing.Options.StartVelocity  := 100;
					gAxBasicPar[AX_X].Homing.Options.HomingVelocity := 30;
					gAxBasicPar[AX_X].Homing.Options.Acceleration   := 150;
					gAxBasicPar[AX_X].Stop.Deceleration			 	:= 2000;
					gAxBasicPar[AX_X].Deceleration					:= 2000;
					gAxBasic[AX_X].Home							:= TRUE;

					gAxBasicPar[AX_Y].Homing.Mode					:= mcHOMING_ABSOLUTE_SWITCH;
					gAxBasicPar[AX_Y].Homing.Options.SensorOffset   := gParameters.LengthParametes.Y_HomeOffsetPos; //gFixData.Ax[AX_X].Config.MultiturnEncOffset; //Home yaptiktan sonra kaçinci pozisyona kadar gitsin
					gAxBasicPar[AX_Y].Homing.Position 			  	:= 0; /gFixData.Ax[AX_X].Par.Homing.Position; //Home yapip Sensor offset kadar gidip bunuda üstüne ekliyor
					gAxBasicPar[AX_Y].Homing.Options.SwitchEdge     := mcDIR_NEGATIVE; //Switch nerede aranacak
					gAxBasicPar[AX_Y].Homing.Options.HomingDirection:= mcDIR_POSITIVE; //switch ten kurtulduktan sonra offset için hangi yöne gidecek
					gAxBasicPar[AX_Y].Homing.Options.StartDirection := mcDIR_NEGATIVE;
					gAxBasicPar[AX_Y].Homing.Options.StartVelocity  := 100;
					gAxBasicPar[AX_Y].Homing.Options.HomingVelocity := 30;
					gAxBasicPar[AX_Y].Homing.Options.Acceleration   := 150;
					gAxBasicPar[AX_Y].Stop.Deceleration			 	:= 2000;
					gAxBasicPar[AX_Y].Deceleration					:= 2000;
					gAxBasic[AX_Y].Home							:= TRUE;

					gAxBasicPar[AX_C].Homing.Mode					:= mcHOMING_ABSOLUTE_SWITCH;
					gAxBasicPar[AX_C].Homing.Options.SensorOffset   := gParameters.LengthParametes.C_HomeOffsetPos; //gFixData.Ax[AX_X].Config.MultiturnEncOffset; //Home yaptiktan sonra kaçinci pozisyona kadar gitsin
					gAxBasicPar[AX_C].Homing.Position 			  	:= 0; /gFixData.Ax[AX_X].Par.Homing.Position; //Home yapip Sensor offset kadar gidip bunuda üstüne ekliyor
					gAxBasicPar[AX_C].Homing.Options.SwitchEdge     := mcDIR_NEGATIVE; //Switch nerede aranacak
					gAxBasicPar[AX_C].Homing.Options.HomingDirection:= mcDIR_POSITIVE; //switch ten kurtulduktan sonra offset için hangi yöne gidecek
					gAxBasicPar[AX_C].Homing.Options.StartDirection := mcDIR_NEGATIVE;
					gAxBasicPar[AX_C].Homing.Options.StartVelocity  := 100;
					gAxBasicPar[AX_C].Homing.Options.HomingVelocity := 30;
					gAxBasicPar[AX_C].Homing.Options.Acceleration   := 150;
					gAxBasicPar[AX_C].Stop.Deceleration			 	:= 2000;
					gAxBasicPar[AX_C].Deceleration					:= 2000;
					gAxBasic[AX_C].Home							:= TRUE;

				ELSE
					IF gMain.Out.Status.Referenced  THEN
						gMain.Out.MainSubStep   	:= SUB_CMD_DONE;
					END_IF;

				END_IF;

		SUB_CMD_DONE:
			IF gMain.Out.Status.Referenced  THEN
				gMain.Out.MainSubStep			:= SUB_INIT;
		//		gMain.Out.MainStep		:= MAIN_WAIT_CMD;
			END_IF;

		SUB_STOP:
			IF Loc.FirstInSubState THEN
				gAxBasic[AX_X].Home			:= FALSE;
				gAxBasic[AX_Y].Home			:= FALSE;
				gAxBasic[AX_C].Home			:= FALSE;
				Loc.Timers.TON_State.IN 	:= FALSE;
			ELSE
				gMain.Out.MainSubStep			:= SUB_INIT;
				//gMain.Out.MainStep		:= MAIN_WAIT_CMD;
			END_IF;

		SUB_ERROR:
			IF Loc.FirstInSubState THEN
				gAxBasic[AX_X].Home			:= FALSE;
				gAxBasic[AX_Y].Home			:= FALSE;
				gAxBasic[AX_C].Home			:= FALSE;
				Loc.Timers.TON_HomeState.IN := FALSE;
			ELSE
				IF gMain.In.Cmd.Reset THEN
					gAxBasic[AX_X].ErrorReset	:= TRUE;
					gAxBasic[AX_Y].ErrorReset	:= TRUE;
					gAxBasic[AX_C].ErrorReset	:= TRUE;
				ELSE
					gAxBasic[AX_X].ErrorReset	:= FALSE;
					gAxBasic[AX_Y].ErrorReset	:= FALSE;
					gAxBasic[AX_C].ErrorReset	:= FALSE;
				END_IF

				IF NOT gAxBasic[AX_X].Error AND NOT gAxBasic[AX_Y].Error NOT gAxBasic[AX_C].Error THEN
					gMain.Out.MainSubStep			:= SUB_INIT;
					//gMain.Out.MainStep		:= MAIN_WAIT_CMD;
				END_IF;

			END_IF;

	END_CASE;

	Loc.Timers.TON_HomeState();

END_ACTION
```
